LIN {X 0,Y 249.072,Z 125.772,A -85,B 0,C 180,E1 -19026.339,E2 -19026.339} C_VEL
LIN {X 0,Y 249.004,Z 125.778,A -85,B 0,C 180,E1 -19030.813,E2 -19030.813} C_VEL
LIN {X 0,Y 250.137,Z 128.804,A -85,B 0,C 180,E1 -19031.188,E2 -19031.188} C_VEL
LIN {X 0,Y 258.788,Z 144.824,A -85,B 0,C 180,E1 -19033.307,E2 -19033.307} C_VEL
LIN {X 0,Y 270.836,Z 168.303,A -85,B 0,C 180,E1 -19036.063,E2 -19036.063} C_VEL
LIN {X 0,Y 280.754,Z 188.589,A -85,B 0,C 180,E1 -19038.178,E2 -19038.178} C_VEL
LIN {X 0,Y 271.037,Z 309.257,A -85,B 0,C 180,E1 -19042.807,E2 -19042.807} C_VEL
LIN {X 0,Y 269.496,Z 326.293,A -85,B 0,C 180,E1 -19043.763,E2 -19043.763} C_VEL
LIN {X 0,Y 267.518,Z 343.702,A -85,B 0,C 180,E1 -19045.037,E2 -19045.037} C_VEL
LIN {X 0,Y 265.194,Z 361.036,A -85,B 0,C 180,E1 -19046.64,E2 -19046.64} C_VEL
LIN {X 0,Y 262.588,Z 377.74,A -85,B 0,C 180,E1 -19048.54,E2 -19048.54} C_VEL
LIN {X 0,Y 259.925,Z 393.091,A -85,B 0,C 180,E1 -19050.654,E2 -19050.654} C_VEL
LIN {X 0,Y 257.421,Z 407.3,A -85,B 0,C 180,E1 -19053.006,E2 -19053.006} C_VEL
LIN {X 0,Y 254.978,Z 420.401,A -85,B 0,C 180,E1 -19055.578,E2 -19055.578} C_VEL
LIN {X 0,Y 252.965,Z 432.478,A -85,B 0,C 180,E1 -19058.4,E2 -19058.4} C_VEL
LIN {X 0,Y 251.134,Z 442.727,A -85,B 0,C 180,E1 -19061.226,E2 -19061.226} C_VEL
LIN {X 0,Y 249.859,Z 451.559,A -85,B 0,C 180,E1 -19064.083,E2 -19064.083} C_VEL
LIN {X 0,Y 248.75,Z 459.037,A -85,B 0,C 180,E1 -19066.937,E2 -19066.937} C_VEL
LIN {X 0,Y 248.058,Z 466.178,A -85,B 0,C 180,E1 -19070.212,E2 -19070.212} C_VEL
LIN {X 0,Y 247.625,Z 471.999,A -85,B 0,C 180,E1 -19073.481,E2 -19073.481} C_VEL
LIN {X 0,Y 247.502,Z 476.6,A -85,B 0,C 180,E1 -19076.744,E2 -19076.744} C_VEL
LIN {X 0,Y 247.516,Z 480.03,A -85,B 0,C 180,E1 -19080,E2 -19080} C_VEL
LIN {X 0,Y 247.605,Z 480.817,A -85,B 0,C 180,E1 -19080.95,E2 -19080.95} C_VEL
LIN {X 0,Y 247.405,Z 481.54,A -85,B 0,C 180,E1 -19081.844,E2 -19081.844} C_VEL
LIN {X 0,Y 245.705,Z 482.796,A -85,B 0,C 180,E1 -19083.616,E2 -19083.616} C_VEL
LIN {X 0,Y 242.493,Z 484.244,A -85,B 0,C 180,E1 -19086.303,E2 -19086.303} C_VEL
LIN {X 0,Y 241.835,Z 484.743,A -85,B 0,C 180,E1 -19087.697,E2 -19087.697} C_VEL
LIN {X 0,Y 241.906,Z 484.875,A -85,B 0,C 180,E1 -19088.165,E2 -19088.165} C_VEL
LIN {X 0,Y 243.543,Z 485.077,A -85,B 0,C 180,E1 -19091.654,E2 -19091.654} C_VEL
LIN {X 0,Y 245.526,Z 484.42,A -85,B 0,C 180,E1 -19094.929,E2 -19094.929} C_VEL
LIN {X 0,Y 248.17,Z 482.778,A -85,B 0,C 180,E1 -19098.15,E2 -19098.15} C_VEL
LIN {X 0,Y 251.479,Z 480.342,A -85,B 0,C 180,E1 -19101.303,E2 -19101.303} C_VEL
LIN {X 0,Y 256.919,Z 475.829,A -85,B 0,C 180,E1 -19105.19,E2 -19105.19} C_VEL
LIN {X 0,Y 263.085,Z 470.156,A -85,B 0,C 180,E1 -19108.741,E2 -19108.741} C_VEL
LIN {X 0,Y 270.575,Z 462.894,A -85,B 0,C 180,E1 -19112.172,E2 -19112.172} C_VEL
LIN {X 0,Y 279.123,Z 454.142,A -85,B 0,C 180,E1 -19115.388,E2 -19115.388} C_VEL
LIN {X 0,Y 288.335,Z 444.274,A -85,B 0,C 180,E1 -19118.206,E2 -19118.206} C_VEL
LIN {X 0,Y 299.61,Z 431.582,A -85,B 0,C 180,E1 -19121.056,E2 -19121.056} C_VEL
LIN {X 0,Y 308.942,Z 420.434,A -85,B 0,C 180,E1 -19123.036,E2 -19123.036} C_VEL
LIN {X 0,Y 310.463,Z 418.647,A -85,B 0,C 180,E1 -19123.581,E2 -19123.581} C_VEL
LIN {X 0,Y 299.973,Z 432.572,A -85,B 0,C 180,E1 -19125.342,E2 -19125.342} C_VEL
LIN {X 0,Y 289.18,Z 446.505,A -85,B 0,C 180,E1 -19127.59,E2 -19127.59} C_VEL
LIN {X 0,Y 279.364,Z 458.973,A -85,B 0,C 180,E1 -19130.095,E2 -19130.095} C_VEL
LIN {X 0,Y 269.8,Z 471.184,A -85,B 0,C 180,E1 -19133.192,E2 -19133.192} C_VEL
LIN {X 0,Y 261.449,Z 481.983,A -85,B 0,C 180,E1 -19136.623,E2 -19136.623} C_VEL
LIN {X 0,Y 255.897,Z 489.259,A -85,B 0,C 180,E1 -19139.462,E2 -19139.462} C_VEL
LIN {X 0,Y 250.118,Z 497.302,A -85,B 0,C 180,E1 -19143.282,E2 -19143.282} C_VEL
LIN {X 0,Y 245.702,Z 503.944,A -85,B 0,C 180,E1 -19147.284,E2 -19147.284} C_VEL
LIN {X 0,Y 242.612,Z 509.118,A -85,B 0,C 180,E1 -19151.418,E2 -19151.418} C_VEL
LIN {X 0,Y 241.094,Z 512.285,A -85,B 0,C 180,E1 -19154.789,E2 -19154.789} C_VEL
LIN {X 0,Y 240.168,Z 514.482,A -85,B 0,C 180,E1 -19158.179,E2 -19158.179} C_VEL
LIN {X 0,Y 240.048,Z 515.814,A -85,B 0,C 180,E1 -19161.581,E2 -19161.581} C_VEL
LIN {X 0,Y 240.331,Z 516.045,A -85,B 0,C 180,E1 -19164.966,E2 -19164.966} C_VEL
LIN {X 0,Y 240.652,Z 515.281,A -85,B 0,C 180,E1 -19168.325,E2 -19168.325} C_VEL
LIN {X 0,Y 240.951,Z 514.432,A -85,B 0,C 180,E1 -19169.999,E2 -19169.999} C_VEL
LIN {X 0,Y 240.777,Z 511.777,A -85,B 0,C 180,E1 -19173.346,E2 -19173.346} C_VEL
LIN {X 0,Y 240.774,Z 507.887,A -85,B 0,C 180,E1 -19176.704,E2 -19176.704} C_VEL
LIN {X 0,Y 240.633,Z 502.482,A -85,B 0,C 180,E1 -19180.091,E2 -19180.091} C_VEL
LIN {X 0,Y 240.972,Z 495.645,A -85,B 0,C 180,E1 -19183.492,E2 -19183.492} C_VEL
LIN {X 0,Y 241.793,Z 487.201,A -85,B 0,C 180,E1 -19186.896,E2 -19186.896} C_VEL
LIN {X 0,Y 242.929,Z 478.349,A -85,B 0,C 180,E1 -19189.871,E2 -19189.871} C_VEL
LIN {X 0,Y 244.802,Z 466.818,A -85,B 0,C 180,E1 -19193.097,E2 -19193.097} C_VEL
LIN {X 0,Y 247.146,Z 453.598,A -85,B 0,C 180,E1 -19196.152,E2 -19196.152} C_VEL
LIN {X 0,Y 249.783,Z 439.422,A -85,B 0,C 180,E1 -19198.866,E2 -19198.866} C_VEL
LIN {X 0,Y 252.637,Z 424.677,A -85,B 0,C 180,E1 -19201.205,E2 -19201.205} C_VEL
LIN {X 0,Y 255.625,Z 408.15,A -85,B 0,C 180,E1 -19203.357,E2 -19203.357} C_VEL
LIN {X 0,Y 258.348,Z 392.121,A -85,B 0,C 180,E1 -19205.057,E2 -19205.057} C_VEL
LIN {X 0,Y 261.07,Z 374.354,A -85,B 0,C 180,E1 -19206.554,E2 -19206.554} C_VEL
LIN {X 0,Y 263.379,Z 357.048,A -85,B 0,C 180,E1 -19207.677,E2 -19207.677} C_VEL
LIN {X 0,Y 265.064,Z 339.199,A -85,B 0,C 180,E1 -19208.541,E2 -19208.541} C_VEL
LIN {X 0,Y 276.313,Z 206.857,A -85,B 0,C 180,E1 -19213.748,E2 -19213.748} C_VEL
LIN {X 0,Y 275.816,Z 204.209,A -85,B 0,C 180,E1 -19213.93,E2 -19213.93} C_VEL
LIN {X 0,Y 262.961,Z 174.544,A -85,B 0,C 180,E1 -19216.972,E2 -19216.972} C_VEL
LIN {X 0,Y 252.135,Z 150.966,A -85,B 0,C 180,E1 -19219.735,E2 -19219.735} C_VEL
LIN {X 0,Y 245.805,Z 137.764,A -85,B 0,C 180,E1 -19221.482,E2 -19221.482} C_VEL
LIN {X 0,Y 242.032,Z 126.649,A -85,B 0,C 180,E1 -19224.497,E2 -19224.497} C_VEL
LIN {X 0,Y 241.972,Z 126.656,A -85,B 0,C 180,E1 -19228.48,E2 -19228.48} C_VEL
LIN {X 0,Y 242.003,Z 126.657,A -85,B 0,C 180,E1 -19232.312,E2 -19232.312} C_VEL
LIN {X 0,Y 242.053,Z 126.649,A -85,B 0,C 180,E1 -19236.016,E2 -19236.016} C_VEL
LIN {X 0,Y 242.033,Z 126.649,A -85,B 0,C 180,E1 -19239.608,E2 -19239.608} C_VEL
LIN {X 0,Y 242.159,Z 126.63,A -85,B 0,C 180,E1 -19243.278,E2 -19243.278} C_VEL
LIN {X 0,Y 242.183,Z 126.624,A -85,B 0,C 180,E1 -19248.28,E2 -19248.28} C_VEL
LIN {X 0,Y 242.431,Z 126.602,A -85,B 0,C 180,E1 -19251.666,E2 -19251.666} C_VEL
LIN {X 0,Y 242.257,Z 126.611,A -85,B 0,C 180,E1 -19255.007,E2 -19255.007} C_VEL
LIN {X 0,Y 242.633,Z 126.573,A -85,B 0,C 180,E1 -19258.34,E2 -19258.34} C_VEL
LIN {X 0,Y 242.633,Z 126.573,A -85,B 0,C 180,E1 -19261.66,E2 -19261.66} C_VEL
LIN {X 0,Y 242.426,Z 126.595,A -85,B 0,C 180,E1 -19266.735,E2 -19266.735} C_VEL
LIN {X 0,Y 242.342,Z 126.608,A -85,B 0,C 180,E1 -19270.021,E2 -19270.021} C_VEL
LIN {X 0,Y 242.163,Z 126.634,A -85,B 0,C 180,E1 -19275.141,E2 -19275.141} C_VEL
LIN {X 0,Y 242.069,Z 126.64,A -85,B 0,C 180,E1 -19278.625,E2 -19278.625} C_VEL
LIN {X 0,Y 242.009,Z 126.649,A -85,B 0,C 180,E1 -19282.18,E2 -19282.18} C_VEL
LIN {X 0,Y 242.063,Z 126.643,A -85,B 0,C 180,E1 -19285.839,E2 -19285.839} C_VEL
LIN {X 0,Y 242.026,Z 126.646,A -85,B 0,C 180,E1 -19289.581,E2 -19289.581} C_VEL
LIN {X 0,Y 241.977,Z 126.655,A -85,B 0,C 180,E1 -19293.493,E2 -19293.493} C_VEL
LIN {X 0,Y 241.985,Z 126.649,A -85,B 0,C 180,E1 -19297.583,E2 -19297.583} C_VEL
LIN {X 0,Y 241.936,Z 126.659,A -85,B 0,C 180,E1 -19301.923,E2 -19301.923} C_VEL
LIN {X 0,Y 241.942,Z 126.654,A -85,B 0,C 180,E1 -19306.569,E2 -19306.569} C_VEL
LIN {X 0,Y 241.986,Z 126.653,A -85,B 0,C 180,E1 -19310.288,E2 -19310.288} C_VEL
LIN {X 0,Y 242.035,Z 126.643,A -85,B 0,C 180,E1 -19314.499,E2 -19314.499} C_VEL
LIN {X 0,Y 241.974,Z 126.657,A -85,B 0,C 180,E1 -19318.481,E2 -19318.481} C_VEL
LIN {X 0,Y 242.005,Z 126.647,A -85,B 0,C 180,E1 -19322.314,E2 -19322.314} C_VEL
LIN {X 0,Y 242.059,Z 126.645,A -85,B 0,C 180,E1 -19326.017,E2 -19326.017} C_VEL
LIN {X 0,Y 242.06,Z 126.64,A -85,B 0,C 180,E1 -19329.611,E2 -19329.611} C_VEL
LIN {X 0,Y 242.163,Z 126.63,A -85,B 0,C 180,E1 -19333.279,E2 -19333.279} C_VEL
LIN {X 0,Y 242.187,Z 126.632,A -85,B 0,C 180,E1 -19338.281,E2 -19338.281} C_VEL
LIN {X 0,Y 242.436,Z 126.594,A -85,B 0,C 180,E1 -19341.667,E2 -19341.667} C_VEL
LIN {X 0,Y 242.261,Z 126.618,A -85,B 0,C 180,E1 -19345.008,E2 -19345.008} C_VEL
LIN {X 0,Y 242.637,Z 126.574,A -85,B 0,C 180,E1 -19348.341,E2 -19348.341} C_VEL
LIN {X 0,Y 242.637,Z 126.571,A -85,B 0,C 180,E1 -19351.661,E2 -19351.661} C_VEL
LIN {X 0,Y 242.436,Z 126.598,A -85,B 0,C 180,E1 -19356.66,E2 -19356.66} C_VEL
LIN {X 0,Y 242.348,Z 126.607,A -85,B 0,C 180,E1 -19360.021,E2 -19360.021} C_VEL
LIN {X 0,Y 242.169,Z 126.633,A -85,B 0,C 180,E1 -19365.142,E2 -19365.142} C_VEL
LIN {X 0,Y 242.076,Z 126.638,A -85,B 0,C 180,E1 -19368.625,E2 -19368.625} C_VEL
LIN {X 0,Y 242.017,Z 126.647,A -85,B 0,C 180,E1 -19372.181,E2 -19372.181} C_VEL
LIN {X 0,Y 242.069,Z 126.645,A -85,B 0,C 180,E1 -19375.839,E2 -19375.839} C_VEL
LIN {X 0,Y 242.032,Z 126.653,A -85,B 0,C 180,E1 -19379.581,E2 -19379.581} C_VEL
LIN {X 0,Y 241.994,Z 126.656,A -85,B 0,C 180,E1 -19383.492,E2 -19383.492} C_VEL
LIN {X 0,Y 242.006,Z 126.65,A -85,B 0,C 180,E1 -19387.58,E2 -19387.58} C_VEL
LIN {X 0,Y 241.947,Z 126.657,A -85,B 0,C 180,E1 -19389.791,E2 -19389.791} C_VEL
LIN {X 0,Y 242.99,Z 129.564,A -85,B 0,C 180,E1 -19390.134,E2 -19390.134} C_VEL
LIN {X 0,Y 244.338,Z 131.856,A -85,B 0,C 180,E1 -19390.479,E2 -19390.479} C_VEL
LIN {X 0,Y 254.963,Z 151.723,A -85,B 0,C 180,E1 -19393.154,E2 -19393.154} C_VEL
LIN {X 0,Y 267.479,Z 176.469,A -85,B 0,C 180,E1 -19396.064,E2 -19396.064} C_VEL
LIN {X 0,Y 274.342,Z 190.869,A -85,B 0,C 180,E1 -19397.576,E2 -19397.576} C_VEL
LIN {X 0,Y 264.433,Z 309.481,A -85,B 0,C 180,E1 -19402.257,E2 -19402.257} C_VEL
LIN {X 0,Y 262.786,Z 327.136,A -85,B 0,C 180,E1 -19403.28,E2 -19403.28} C_VEL
LIN {X 0,Y 260.733,Z 344.437,A -85,B 0,C 180,E1 -19404.583,E2 -19404.583} C_VEL
LIN {X 0,Y 258.512,Z 360.775,A -85,B 0,C 180,E1 -19406.129,E2 -19406.129} C_VEL
LIN {X 0,Y 255.822,Z 377.614,A -85,B 0,C 180,E1 -19408.073,E2 -19408.073} C_VEL
LIN {X 0,Y 253.1,Z 393.039,A -85,B 0,C 180,E1 -19410.241,E2 -19410.241} C_VEL
LIN {X 0,Y 250.503,Z 407.312,A -85,B 0,C 180,E1 -19412.651,E2 -19412.651} C_VEL
LIN {X 0,Y 247.9,Z 421.11,A -85,B 0,C 180,E1 -19415.426,E2 -19415.426} C_VEL
LIN {X 0,Y 245.912,Z 432.635,A -85,B 0,C 180,E1 -19418.19,E2 -19418.19} C_VEL
LIN {X 0,Y 244.055,Z 442.978,A -85,B 0,C 180,E1 -19421.097,E2 -19421.097} C_VEL
LIN {X 0,Y 242.733,Z 451.861,A -85,B 0,C 180,E1 -19424.034,E2 -19424.034} C_VEL
LIN {X 0,Y 241.529,Z 460.386,A -85,B 0,C 180,E1 -19427.394,E2 -19427.394} C_VEL
LIN {X 0,Y 240.858,Z 467.389,A -85,B 0,C 180,E1 -19430.765,E2 -19430.765} C_VEL
LIN {X 0,Y 240.452,Z 473.046,A -85,B 0,C 180,E1 -19434.11,E2 -19434.11} C_VEL
LIN {X 0,Y 240.426,Z 476.555,A -85,B 0,C 180,E1 -19436.648,E2 -19436.648} C_VEL
LIN {X 0,Y 240.425,Z 480.217,A -85,B 0,C 180,E1 -19440,E2 -19440} C_VEL
LIN {X 0,Y 240.885,Z 482.815,A -85,B 0,C 180,E1 -19443.345,E2 -19443.345} C_VEL
LIN {X 0,Y 241.482,Z 484.438,A -85,B 0,C 180,E1 -19446.685,E2 -19446.685} C_VEL
LIN {X 0,Y 241.906,Z 484.875,A -85,B 0,C 180,E1 -19448.165,E2 -19448.165} C_VEL
LIN {X 0,Y 241.779,Z 485.264,A -85,B 0,C 180,E1 -19449.562,E2 -19449.562} C_VEL
LIN {X 0,Y 240.042,Z 485.702,A -85,B 0,C 180,E1 -19451.882,E2 -19451.882} C_VEL
LIN {X 0,Y 238.742,Z 485.726,A -85,B 0,C 180,E1 -19453.762,E2 -19453.762} C_VEL
LIN {X 0,Y 238.672,Z 485.475,A -85,B 0,C 180,E1 -19455.183,E2 -19455.183} C_VEL
LIN {X 0,Y 238.933,Z 485.329,A -85,B 0,C 180,E1 -19455.652,E2 -19455.652} C_VEL
LIN {X 0,Y 243.189,Z 483.096,A -85,B 0,C 180,E1 -19460.291,E2 -19460.291} C_VEL
LIN {X 0,Y 247.128,Z 480.38,A -85,B 0,C 180,E1 -19463.462,E2 -19463.462} C_VEL
LIN {X 0,Y 253.4,Z 475.577,A -85,B 0,C 180,E1 -19467.435,E2 -19467.435} C_VEL
LIN {X 0,Y 260.197,Z 469.904,A -85,B 0,C 180,E1 -19470.877,E2 -19470.877} C_VEL
LIN {X 0,Y 268.479,Z 462.552,A -85,B 0,C 180,E1 -19474.25,E2 -19474.25} C_VEL
LIN {X 0,Y 277.871,Z 453.719,A -85,B 0,C 180,E1 -19477.374,E2 -19477.374} C_VEL
LIN {X 0,Y 287.282,Z 444.421,A -85,B 0,C 180,E1 -19479.954,E2 -19479.954} C_VEL
LIN {X 0,Y 298.648,Z 432.545,A -85,B 0,C 180,E1 -19482.576,E2 -19482.576} C_VEL
LIN {X 0,Y 301.527,Z 429.387,A -85,B 0,C 180,E1 -19483.167,E2 -19483.167} C_VEL
LIN {X 0,Y 300.71,Z 430.48,A -85,B 0,C 180,E1 -19483.571,E2 -19483.571} C_VEL
LIN {X 0,Y 289.203,Z 444.239,A -85,B 0,C 180,E1 -19485.679,E2 -19485.679} C_VEL
LIN {X 0,Y 278.639,Z 456.594,A -85,B 0,C 180,E1 -19488.055,E2 -19488.055} C_VEL
LIN {X 0,Y 269.174,Z 467.539,A -85,B 0,C 180,E1 -19490.715,E2 -19490.715} C_VEL
LIN {X 0,Y 259.872,Z 478.33,A -85,B 0,C 180,E1 -19493.969,E2 -19493.969} C_VEL
LIN {X 0,Y 252.646,Z 486.874,A -85,B 0,C 180,E1 -19497.149,E2 -19497.149} C_VEL
LIN {X 0,Y 246.081,Z 495.016,A -85,B 0,C 180,E1 -19500.953,E2 -19500.953} C_VEL
LIN {X 0,Y 241.207,Z 501.217,A -85,B 0,C 180,E1 -19504.587,E2 -19504.587} C_VEL
LIN {X 0,Y 236.913,Z 507.236,A -85,B 0,C 180,E1 -19509.145,E2 -19509.145} C_VEL
LIN {X 0,Y 234.429,Z 511.459,A -85,B 0,C 180,E1 -19513.603,E2 -19513.603} C_VEL
LIN {X 0,Y 233.137,Z 514.042,A -85,B 0,C 180,E1 -19517.817,E2 -19517.817} C_VEL
LIN {X 0,Y 232.96,Z 515.129,A -85,B 0,C 180,E1 -19521.323,E2 -19521.323} C_VEL
LIN {X 0,Y 233.27,Z 515.257,A -85,B 0,C 180,E1 -19524.813,E2 -19524.813} C_VEL
LIN {X 0,Y 233.636,Z 514.3,A -85,B 0,C 180,E1 -19528.275,E2 -19528.275} C_VEL
LIN {X 0,Y 233.913,Z 513.44,A -85,B 0,C 180,E1 -19529.999,E2 -19529.999} C_VEL
LIN {X 0,Y 233.753,Z 510.574,A -85,B 0,C 180,E1 -19533.446,E2 -19533.446} C_VEL
LIN {X 0,Y 233.747,Z 506.487,A -85,B 0,C 180,E1 -19536.906,E2 -19536.906} C_VEL
LIN {X 0,Y 233.617,Z 500.93,A -85,B 0,C 180,E1 -19540.398,E2 -19540.398} C_VEL
LIN {X 0,Y 234.009,Z 493.845,A -85,B 0,C 180,E1 -19543.901,E2 -19543.901} C_VEL
LIN {X 0,Y 234.905,Z 485.132,A -85,B 0,C 180,E1 -19547.407,E2 -19547.407} C_VEL
LIN {X 0,Y 236.107,Z 475.965,A -85,B 0,C 180,E1 -19550.471,E2 -19550.471} C_VEL
LIN {X 0,Y 237.947,Z 465.069,A -85,B 0,C 180,E1 -19553.536,E2 -19553.536} C_VEL
LIN {X 0,Y 240.244,Z 452.502,A -85,B 0,C 180,E1 -19556.493,E2 -19556.493} C_VEL
LIN {X 0,Y 242.677,Z 439.747,A -85,B 0,C 180,E1 -19559.017,E2 -19559.017} C_VEL
LIN {X 0,Y 245.628,Z 424.816,A -85,B 0,C 180,E1 -19561.477,E2 -19561.477} C_VEL
LIN {X 0,Y 248.653,Z 408.492,A -85,B 0,C 180,E1 -19563.688,E2 -19563.688} C_VEL
LIN {X 0,Y 251.446,Z 392.494,A -85,B 0,C 180,E1 -19565.447,E2 -19565.447} C_VEL
LIN {X 0,Y 254.246,Z 374.872,A -85,B 0,C 180,E1 -19566.992,E2 -19566.992} C_VEL
LIN {X 0,Y 256.732,Z 356.781,A -85,B 0,C 180,E1 -19568.205,E2 -19568.205} C_VEL
LIN {X 0,Y 258.446,Z 339.216,A -85,B 0,C 180,E1 -19569.089,E2 -19569.089} C_VEL
LIN {X 0,Y 270.009,Z 207.635,A -85,B 0,C 180,E1 -19574.425,E2 -19574.425} C_VEL
LIN {X 0,Y 257.52,Z 178.451,A -85,B 0,C 180,E1 -19577.486,E2 -19577.486} C_VEL
LIN {X 0,Y 245.86,Z 153.121,A -85,B 0,C 180,E1 -19580.544,E2 -19580.544} C_VEL
LIN {X 0,Y 238.279,Z 137.255,A -85,B 0,C 180,E1 -19582.705,E2 -19582.705} C_VEL
LIN {X 0,Y 234.94,Z 127.532,A -85,B 0,C 180,E1 -19585.417,E2 -19585.417} C_VEL
LIN {X 0,Y 234.928,Z 127.535,A -85,B 0,C 180,E1 -19589.432,E2 -19589.432} C_VEL
LIN {X 0,Y 234.99,Z 127.528,A -85,B 0,C 180,E1 -19593.793,E2 -19593.793} C_VEL
LIN {X 0,Y 235.007,Z 127.524,A -85,B 0,C 180,E1 -19598.97,E2 -19598.97} C_VEL
LIN {X 0,Y 235.092,Z 127.51,A -85,B 0,C 180,E1 -19603.059,E2 -19603.059} C_VEL
LIN {X 0,Y 235.143,Z 127.5,A -85,B 0,C 180,E1 -19607.924,E2 -19607.924} C_VEL
LIN {X 0,Y 235.386,Z 127.478,A -85,B 0,C 180,E1 -19611.415,E2 -19611.415} C_VEL
LIN {X 0,Y 235.402,Z 127.473,A -85,B 0,C 180,E1 -19613.141,E2 -19613.141} C_VEL
LIN {X 0,Y 235.592,Z 127.451,A -85,B 0,C 180,E1 -19618.291,E2 -19618.291} C_VEL
LIN {X 0,Y 235.592,Z 127.45,A -85,B 0,C 180,E1 -19621.71,E2 -19621.71} C_VEL
LIN {X 0,Y 235.402,Z 127.471,A -85,B 0,C 180,E1 -19626.859,E2 -19626.859} C_VEL
LIN {X 0,Y 235.249,Z 127.491,A -85,B 0,C 180,E1 -19630.326,E2 -19630.326} C_VEL
LIN {X 0,Y 235.11,Z 127.51,A -85,B 0,C 180,E1 -19635.607,E2 -19635.607} C_VEL
LIN {X 0,Y 235.005,Z 127.523,A -85,B 0,C 180,E1 -19639.206,E2 -19639.206} C_VEL
LIN {X 0,Y 234.957,Z 127.529,A -85,B 0,C 180,E1 -19642.883,E2 -19642.883} C_VEL
LIN {X 0,Y 234.966,Z 127.527,A -85,B 0,C 180,E1 -19646.658,E2 -19646.658} C_VEL
LIN {X 0,Y 234.928,Z 127.53,A -85,B 0,C 180,E1 -19650.568,E2 -19650.568} C_VEL
LIN {X 0,Y 234.926,Z 127.534,A -85,B 0,C 180,E1 -19654.639,E2 -19654.639} C_VEL
LIN {X 0,Y 234.938,Z 127.527,A -85,B 0,C 180,E1 -19658.945,E2 -19658.945} C_VEL
LIN {X 0,Y 234.888,Z 127.537,A -85,B 0,C 180,E1 -19663.486,E2 -19663.486} C_VEL
LIN {X 0,Y 234.92,Z 127.529,A -85,B 0,C 180,E1 -19666.523,E2 -19666.523} C_VEL
LIN {X 0,Y 234.952,Z 127.529,A -85,B 0,C 180,E1 -19671.087,E2 -19671.087} C_VEL
LIN {X 0,Y 234.959,Z 127.526,A -85,B 0,C 180,E1 -19675.368,E2 -19675.368} C_VEL
LIN {X 0,Y 234.967,Z 127.527,A -85,B 0,C 180,E1 -19680.159,E2 -19680.159} C_VEL
LIN {X 0,Y 234.993,Z 127.523,A -85,B 0,C 180,E1 -19683.795,E2 -19683.795} C_VEL
LIN {X 0,Y 235.027,Z 127.517,A -85,B 0,C 180,E1 -19688.973,E2 -19688.973} C_VEL
LIN {X 0,Y 235.096,Z 127.511,A -85,B 0,C 180,E1 -19693.06,E2 -19693.06} C_VEL
LIN {X 0,Y 235.119,Z 127.51,A -85,B 0,C 180,E1 -19697.923,E2 -19697.923} C_VEL
LIN {X 0,Y 235.391,Z 127.47,A -85,B 0,C 180,E1 -19701.416,E2 -19701.416} C_VEL
LIN {X 0,Y 235.406,Z 127.472,A -85,B 0,C 180,E1 -19703.143,E2 -19703.143} C_VEL
LIN {X 0,Y 235.597,Z 127.452,A -85,B 0,C 180,E1 -19708.292,E2 -19708.292} C_VEL
LIN {X 0,Y 235.597,Z 127.447,A -85,B 0,C 180,E1 -19711.711,E2 -19711.711} C_VEL
LIN {X 0,Y 235.407,Z 127.473,A -85,B 0,C 180,E1 -19716.86,E2 -19716.86} C_VEL
LIN {X 0,Y 235.255,Z 127.488,A -85,B 0,C 180,E1 -19720.327,E2 -19720.327} C_VEL
LIN {X 0,Y 235.116,Z 127.514,A -85,B 0,C 180,E1 -19725.607,E2 -19725.607} C_VEL
LIN {X 0,Y 235.012,Z 127.518,A -85,B 0,C 180,E1 -19729.206,E2 -19729.206} C_VEL
LIN {X 0,Y 234.965,Z 127.524,A -85,B 0,C 180,E1 -19732.884,E2 -19732.884} C_VEL
LIN {X 0,Y 234.972,Z 127.527,A -85,B 0,C 180,E1 -19736.658,E2 -19736.658} C_VEL
LIN {X 0,Y 234.935,Z 127.533,A -85,B 0,C 180,E1 -19740.569,E2 -19740.569} C_VEL
LIN {X 0,Y 234.964,Z 127.527,A -85,B 0,C 180,E1 -19744.634,E2 -19744.634} C_VEL
LIN {X 0,Y 234.947,Z 127.559,A -85,B 0,C 180,E1 -19748.72,E2 -19748.72} C_VEL
LIN {X 0,Y 235.955,Z 130.389,A -85,B 0,C 180,E1 -19749.062,E2 -19749.062} C_VEL
LIN {X 0,Y 244.618,Z 146.212,A -85,B 0,C 180,E1 -19751.362,E2 -19751.362} C_VEL
LIN {X 0,Y 257.248,Z 170.753,A -85,B 0,C 180,E1 -19754.486,E2 -19754.486} C_VEL
LIN {X 0,Y 267.827,Z 192.409,A -85,B 0,C 180,E1 -19756.899,E2 -19756.899} C_VEL
LIN {X 0,Y 265.441,Z 220.63,A -85,B 0,C 180,E1 -19758.024,E2 -19758.024} C_VEL
LIN {X 0,Y 257.797,Z 310.244,A -85,B 0,C 180,E1 -19761.719,E2 -19761.719} C_VEL
LIN {X 0,Y 256.17,Z 326.998,A -85,B 0,C 180,E1 -19762.715,E2 -19762.715} C_VEL
LIN {X 0,Y 253.984,Z 345.031,A -85,B 0,C 180,E1 -19764.106,E2 -19764.106} C_VEL
LIN {X 0,Y 251.537,Z 362.229,A -85,B 0,C 180,E1 -19765.785,E2 -19765.785} C_VEL
LIN {X 0,Y 248.775,Z 379.205,A -85,B 0,C 180,E1 -19767.829,E2 -19767.829} C_VEL
LIN {X 0,Y 246.01,Z 394.186,A -85,B 0,C 180,E1 -19770.004,E2 -19770.004} C_VEL
LIN {X 0,Y 243.379,Z 408.38,A -85,B 0,C 180,E1 -19772.482,E2 -19772.482} C_VEL
LIN {X 0,Y 240.929,Z 421.124,A -85,B 0,C 180,E1 -19775.126,E2 -19775.126} C_VEL
LIN {X 0,Y 238.886,Z 432.733,A -85,B 0,C 180,E1 -19777.969,E2 -19777.969} C_VEL
LIN {X 0,Y 236.837,Z 444.198,A -85,B 0,C 180,E1 -19781.294,E2 -19781.294} C_VEL
LIN {X 0,Y 235.411,Z 453.238,A -85,B 0,C 180,E1 -19784.414,E2 -19784.414} C_VEL
LIN {X 0,Y 234.316,Z 461.645,A -85,B 0,C 180,E1 -19787.88,E2 -19787.88} C_VEL
LIN {X 0,Y 233.717,Z 468.561,A -85,B 0,C 180,E1 -19791.352,E2 -19791.352} C_VEL
LIN {X 0,Y 233.342,Z 474.121,A -85,B 0,C 180,E1 -19794.816,E2 -19794.816} C_VEL
LIN {X 0,Y 233.288,Z 478.56,A -85,B 0,C 180,E1 -19798.273,E2 -19798.273} C_VEL
LIN {X 0,Y 233.53,Z 481.851,A -85,B 0,C 180,E1 -19801.724,E2 -19801.724} C_VEL
LIN {X 0,Y 234.096,Z 484.152,A -85,B 0,C 180,E1 -19805.167,E2 -19805.167} C_VEL
LIN {X 0,Y 234.967,Z 485.508,A -85,B 0,C 180,E1 -19808.601,E2 -19808.601} C_VEL
LIN {X 0,Y 236.623,Z 485.909,A -85,B 0,C 180,E1 -19812,E2 -19812} C_VEL
LIN {X 0,Y 238.933,Z 485.329,A -85,B 0,C 180,E1 -19815.652,E2 -19815.652} C_VEL
LIN {X 0,Y 239.382,Z 484.966,A -85,B 0,C 180,E1 -19817.061,E2 -19817.061} C_VEL
LIN {X 0,Y 238.676,Z 484.454,A -85,B 0,C 180,E1 -19819.432,E2 -19819.432} C_VEL
LIN {X 0,Y 238.397,Z 483.717,A -85,B 0,C 180,E1 -19821.803,E2 -19821.803} C_VEL
LIN {X 0,Y 239.491,Z 482.826,A -85,B 0,C 180,E1 -19823.176,E2 -19823.176} C_VEL
LIN {X 0,Y 245.746,Z 478.777,A -85,B 0,C 180,E1 -19827.231,E2 -19827.231} C_VEL
LIN {X 0,Y 252.964,Z 473.532,A -85,B 0,C 180,E1 -19830.929,E2 -19830.929} C_VEL
LIN {X 0,Y 261.329,Z 466.956,A -85,B 0,C 180,E1 -19834.385,E2 -19834.385} C_VEL
LIN {X 0,Y 270.832,Z 458.986,A -85,B 0,C 180,E1 -19837.576,E2 -19837.576} C_VEL
LIN {X 0,Y 281.474,Z 449.55,A -85,B 0,C 180,E1 -19840.48,E2 -19840.48} C_VEL
LIN {X 0,Y 292.923,Z 438.77,A -85,B 0,C 180,E1 -19843.052,E2 -19843.052} C_VEL
LIN {X 0,Y 292.366,Z 439.463,A -85,B 0,C 180,E1 -19843.341,E2 -19843.341} C_VEL
LIN {X 0,Y 280.864,Z 451.884,A -85,B 0,C 180,E1 -19845.521,E2 -19845.521} C_VEL
LIN {X 0,Y 269.258,Z 464.188,A -85,B 0,C 180,E1 -19848.272,E2 -19848.272} C_VEL
LIN {X 0,Y 259.008,Z 475.066,A -85,B 0,C 180,E1 -19851.384,E2 -19851.384} C_VEL
LIN {X 0,Y 248.336,Z 486.343,A -85,B 0,C 180,E1 -19855.527,E2 -19855.527} C_VEL
LIN {X 0,Y 241.186,Z 494.322,A -85,B 0,C 180,E1 -19859.339,E2 -19859.339} C_VEL
LIN {X 0,Y 235.307,Z 500.964,A -85,B 0,C 180,E1 -19863.383,E2 -19863.383} C_VEL
LIN {X 0,Y 231.691,Z 505.408,A -85,B 0,C 180,E1 -19866.774,E2 -19866.774} C_VEL
LIN {X 0,Y 228.004,Z 510.443,A -85,B 0,C 180,E1 -19872.046,E2 -19872.046} C_VEL
LIN {X 0,Y 226.565,Z 512.697,A -85,B 0,C 180,E1 -19875.63,E2 -19875.63} C_VEL
LIN {X 0,Y 225.901,Z 514.124,A -85,B 0,C 180,E1 -19879.241,E2 -19879.241} C_VEL
LIN {X 0,Y 226.151,Z 514.504,A -85,B 0,C 180,E1 -19883.959,E2 -19883.959} C_VEL
LIN {X 0,Y 226.419,Z 514,A -85,B 0,C 180,E1 -19886.44,E2 -19886.44} C_VEL
LIN {X 0,Y 226.892,Z 512.325,A -85,B 0,C 180,E1 -19889.999,E2 -19889.999} C_VEL
LIN {X 0,Y 226.81,Z 511.019,A -85,B 0,C 180,E1 -19891.774,E2 -19891.774} C_VEL
LIN {X 0,Y 226.725,Z 507.356,A -85,B 0,C 180,E1 -19895.335,E2 -19895.335} C_VEL
LIN {X 0,Y 226.643,Z 503.871,A -85,B 0,C 180,E1 -19897.93,E2 -19897.93} C_VEL
LIN {X 0,Y 226.651,Z 497.553,A -85,B 0,C 180,E1 -19901.627,E2 -19901.627} C_VEL
LIN {X 0,Y 227.248,Z 489.864,A -85,B 0,C 180,E1 -19905.24,E2 -19905.24} C_VEL
LIN {X 0,Y 228.354,Z 480.411,A -85,B 0,C 180,E1 -19908.853,E2 -19908.853} C_VEL
LIN {X 0,Y 229.838,Z 470.538,A -85,B 0,C 180,E1 -19911.997,E2 -19911.997} C_VEL
LIN {X 0,Y 231.899,Z 458.922,A -85,B 0,C 180,E1 -19915.104,E2 -19915.104} C_VEL
LIN {X 0,Y 234.58,Z 445.191,A -85,B 0,C 180,E1 -19918.154,E2 -19918.154} C_VEL
LIN {X 0,Y 237.238,Z 431.741,A -85,B 0,C 180,E1 -19920.65,E2 -19920.65} C_VEL
LIN {X 0,Y 240.258,Z 416.361,A -85,B 0,C 180,E1 -19923.011,E2 -19923.011} C_VEL
LIN {X 0,Y 243.294,Z 400.229,A -85,B 0,C 180,E1 -19925.037,E2 -19925.037} C_VEL
LIN {X 0,Y 246.255,Z 382.596,A -85,B 0,C 180,E1 -19926.82,E2 -19926.82} C_VEL
LIN {X 0,Y 248.768,Z 365.826,A -85,B 0,C 180,E1 -19928.153,E2 -19928.153} C_VEL
LIN {X 0,Y 251.033,Z 347.901,A -85,B 0,C 180,E1 -19929.236,E2 -19929.236} C_VEL
LIN {X 0,Y 262.28,Z 223.969,A -85,B 0,C 180,E1 -19934.496,E2 -19934.496} C_VEL
LIN {X 0,Y 263.554,Z 209.377,A -85,B 0,C 180,E1 -19935.096,E2 -19935.096} C_VEL
LIN {X 0,Y 251.763,Z 181.744,A -85,B 0,C 180,E1 -19938.069,E2 -19938.069} C_VEL
LIN {X 0,Y 240.894,Z 157.856,A -85,B 0,C 180,E1 -19941.018,E2 -19941.018} C_VEL
LIN {X 0,Y 230.756,Z 136.797,A -85,B 0,C 180,E1 -19943.972,E2 -19943.972} C_VEL
LIN {X 0,Y 227.911,Z 128.407,A -85,B 0,C 180,E1 -19946.435,E2 -19946.435} C_VEL
LIN {X 0,Y 227.914,Z 128.409,A -85,B 0,C 180,E1 -19950.437,E2 -19950.437} C_VEL
LIN {X 0,Y 227.924,Z 128.412,A -85,B 0,C 180,E1 -19954.426,E2 -19954.426} C_VEL
LIN {X 0,Y 227.958,Z 128.405,A -85,B 0,C 180,E1 -19958.287,E2 -19958.287} C_VEL
LIN {X 0,Y 228.031,Z 128.389,A -85,B 0,C 180,E1 -19962.825,E2 -19962.825} C_VEL
LIN {X 0,Y 228.09,Z 128.378,A -85,B 0,C 180,E1 -19967.544,E2 -19967.544} C_VEL
LIN {X 0,Y 228.321,Z 128.357,A -85,B 0,C 180,E1 -19971.147,E2 -19971.147} C_VEL
LIN {X 0,Y 228.354,Z 128.351,A -85,B 0,C 180,E1 -19972.929,E2 -19972.929} C_VEL
LIN {X 0,Y 228.551,Z 128.328,A -85,B 0,C 180,E1 -19978.238,E2 -19978.238} C_VEL
LIN {X 0,Y 228.551,Z 128.327,A -85,B 0,C 180,E1 -19981.762,E2 -19981.762} C_VEL
LIN {X 0,Y 228.355,Z 128.349,A -85,B 0,C 180,E1 -19987.072,E2 -19987.072} C_VEL
LIN {X 0,Y 228.168,Z 128.373,A -85,B 0,C 180,E1 -19990.65,E2 -19990.65} C_VEL
LIN {X 0,Y 228.054,Z 128.387,A -85,B 0,C 180,E1 -19996.103,E2 -19996.103} C_VEL
LIN {X 0,Y 227.939,Z 128.404,A -85,B 0,C 180,E1 -19999.826,E2 -19999.826} C_VEL
LIN {X 0,Y 227.91,Z 128.401,A -85,B 0,C 180,E1 -20003.633,E2 -20003.633} C_VEL
LIN {X 0,Y 227.882,Z 128.411,A -85,B 0,C 180,E1 -20007.556,E2 -20007.556} C_VEL
LIN {X 0,Y 227.867,Z 128.408,A -85,B 0,C 180,E1 -20011.623,E2 -20011.623} C_VEL
LIN {X 0,Y 227.877,Z 128.41,A -85,B 0,C 180,E1 -20015.873,E2 -20015.873} C_VEL
LIN {X 0,Y 227.823,Z 128.414,A -85,B 0,C 180,E1 -20020.377,E2 -20020.377} C_VEL
LIN {X 0,Y 227.835,Z 128.411,A -85,B 0,C 180,E1 -20025.192,E2 -20025.192} C_VEL
LIN {X 0,Y 227.872,Z 128.411,A -85,B 0,C 180,E1 -20029.635,E2 -20029.635} C_VEL
LIN {X 0,Y 227.899,Z 128.402,A -85,B 0,C 180,E1 -20034.133,E2 -20034.133} C_VEL
LIN {X 0,Y 227.871,Z 128.413,A -85,B 0,C 180,E1 -20038.379,E2 -20038.379} C_VEL
LIN {X 0,Y 227.884,Z 128.406,A -85,B 0,C 180,E1 -20042.446,E2 -20042.446} C_VEL
LIN {X 0,Y 227.924,Z 128.407,A -85,B 0,C 180,E1 -20046.37,E2 -20046.37} C_VEL
LIN {X 0,Y 227.954,Z 128.399,A -85,B 0,C 180,E1 -20050.177,E2 -20050.177} C_VEL
LIN {X 0,Y 228.058,Z 128.389,A -85,B 0,C 180,E1 -20053.899,E2 -20053.899} C_VEL
LIN {X 0,Y 228.076,Z 128.386,A -85,B 0,C 180,E1 -20057.545,E2 -20057.545} C_VEL
LIN {X 0,Y 228.326,Z 128.35,A -85,B 0,C 180,E1 -20061.148,E2 -20061.148} C_VEL
LIN {X 0,Y 228.359,Z 128.35,A -85,B 0,C 180,E1 -20062.93,E2 -20062.93} C_VEL
LIN {X 0,Y 228.555,Z 128.328,A -85,B 0,C 180,E1 -20068.239,E2 -20068.239} C_VEL
LIN {X 0,Y 228.555,Z 128.323,A -85,B 0,C 180,E1 -20071.763,E2 -20071.763} C_VEL
LIN {X 0,Y 228.36,Z 128.352,A -85,B 0,C 180,E1 -20077.072,E2 -20077.072} C_VEL
LIN {X 0,Y 228.174,Z 128.369,A -85,B 0,C 180,E1 -20080.651,E2 -20080.651} C_VEL
LIN {X 0,Y 228.06,Z 128.389,A -85,B 0,C 180,E1 -20086.103,E2 -20086.103} C_VEL
LIN {X 0,Y 227.946,Z 128.403,A -85,B 0,C 180,E1 -20089.826,E2 -20089.826} C_VEL
LIN {X 0,Y 227.917,Z 128.402,A -85,B 0,C 180,E1 -20093.633,E2 -20093.633} C_VEL
LIN {X 0,Y 227.888,Z 128.408,A -85,B 0,C 180,E1 -20097.556,E2 -20097.556} C_VEL
LIN {X 0,Y 227.876,Z 128.41,A -85,B 0,C 180,E1 -20101.623,E2 -20101.623} C_VEL
LIN {X 0,Y 227.903,Z 128.41,A -85,B 0,C 180,E1 -20105.869,E2 -20105.869} C_VEL
LIN {X 0,Y 227.942,Z 128.468,A -85,B 0,C 180,E1 -20107.591,E2 -20107.591} C_VEL
LIN {X 0,Y 228.933,Z 131.264,A -85,B 0,C 180,E1 -20107.945,E2 -20107.945} C_VEL
LIN {X 0,Y 238.918,Z 149.481,A -85,B 0,C 180,E1 -20110.697,E2 -20110.697} C_VEL
LIN {X 0,Y 252.24,Z 175.591,A -85,B 0,C 180,E1 -20114.088,E2 -20114.088} C_VEL
LIN {X 0,Y 261.487,Z 194.703,A -85,B 0,C 180,E1 -20116.265,E2 -20116.265} C_VEL
LIN {X 0,Y 251.224,Z 310.134,A -85,B 0,C 180,E1 -20121.12,E2 -20121.12} C_VEL
LIN {X 0,Y 249.523,Z 327.21,A -85,B 0,C 180,E1 -20122.158,E2 -20122.158} C_VEL
LIN {X 0,Y 247.24,Z 345.49,A -85,B 0,C 180,E1 -20123.602,E2 -20123.602} C_VEL
LIN {X 0,Y 244.577,Z 363.516,A -85,B 0,C 180,E1 -20125.422,E2 -20125.422} C_VEL
LIN {X 0,Y 241.918,Z 379.499,A -85,B 0,C 180,E1 -20127.405,E2 -20127.405} C_VEL
LIN {X 0,Y 238.971,Z 395.206,A -85,B 0,C 180,E1 -20129.759,E2 -20129.759} C_VEL
LIN {X 0,Y 236.304,Z 409.343,A -85,B 0,C 180,E1 -20132.309,E2 -20132.309} C_VEL
LIN {X 0,Y 233.744,Z 422.386,A -85,B 0,C 180,E1 -20135.106,E2 -20135.106} C_VEL
LIN {X 0,Y 231.856,Z 432.775,A -85,B 0,C 180,E1 -20137.734,E2 -20137.734} C_VEL
LIN {X 0,Y 229.743,Z 444.399,A -85,B 0,C 180,E1 -20141.187,E2 -20141.187} C_VEL
LIN {X 0,Y 228.326,Z 453.436,A -85,B 0,C 180,E1 -20144.375,E2 -20144.375} C_VEL
LIN {X 0,Y 227.304,Z 460.921,A -85,B 0,C 180,E1 -20147.5,E2 -20147.5} C_VEL
LIN {X 0,Y 226.64,Z 468.057,A -85,B 0,C 180,E1 -20151.08,E2 -20151.08} C_VEL
LIN {X 0,Y 226.257,Z 473.894,A -85,B 0,C 180,E1 -20154.653,E2 -20154.653} C_VEL
LIN {X 0,Y 226.209,Z 478.518,A -85,B 0,C 180,E1 -20158.219,E2 -20158.219} C_VEL
LIN {X 0,Y 226.445,Z 481.999,A -85,B 0,C 180,E1 -20161.778,E2 -20161.778} C_VEL
LIN {X 0,Y 227.039,Z 484.546,A -85,B 0,C 180,E1 -20165.328,E2 -20165.328} C_VEL
LIN {X 0,Y 228.706,Z 486.48,A -85,B 0,C 180,E1 -20170.468,E2 -20170.468} C_VEL
LIN {X 0,Y 230.736,Z 486.67,A -85,B 0,C 180,E1 -20174.103,E2 -20174.103} C_VEL
LIN {X 0,Y 233.329,Z 486,A -85,B 0,C 180,E1 -20177.53,E2 -20177.53} C_VEL
LIN {X 0,Y 236.67,Z 484.432,A -85,B 0,C 180,E1 -20180.876,E2 -20180.876} C_VEL
LIN {X 0,Y 239.491,Z 482.826,A -85,B 0,C 180,E1 -20183.176,E2 -20183.176} C_VEL
LIN {X 0,Y 240.751,Z 481.921,A -85,B 0,C 180,E1 -20184.538,E2 -20184.538} C_VEL
LIN {X 0,Y 242.217,Z 479.518,A -85,B 0,C 180,E1 -20188.723,E2 -20188.723} C_VEL
LIN {X 0,Y 243.675,Z 478.265,A -85,B 0,C 180,E1 -20190.037,E2 -20190.037} C_VEL
LIN {X 0,Y 244.426,Z 477.738,A -85,B 0,C 180,E1 -20190.445,E2 -20190.445} C_VEL
LIN {X 0,Y 252.349,Z 472.398,A -85,B 0,C 180,E1 -20193.849,E2 -20193.849} C_VEL
LIN {X 0,Y 261.755,Z 465.5,A -85,B 0,C 180,E1 -20197.165,E2 -20197.165} C_VEL
LIN {X 0,Y 272.308,Z 457.23,A -85,B 0,C 180,E1 -20200.182,E2 -20200.182} C_VEL
LIN {X 0,Y 281.529,Z 449.571,A -85,B 0,C 180,E1 -20202.378,E2 -20202.378} C_VEL
LIN {X 0,Y 283.506,Z 448.027,A -85,B 0,C 180,E1 -20203.178,E2 -20203.178} C_VEL
LIN {X 0,Y 271.308,Z 460.03,A -85,B 0,C 180,E1 -20205.619,E2 -20205.619} C_VEL
LIN {X 0,Y 259.917,Z 470.98,A -85,B 0,C 180,E1 -20208.511,E2 -20208.511} C_VEL
LIN {X 0,Y 249.83,Z 480.687,A -85,B 0,C 180,E1 -20211.764,E2 -20211.764} C_VEL
LIN {X 0,Y 241.011,Z 489.216,A -85,B 0,C 180,E1 -20215.344,E2 -20215.344} C_VEL
LIN {X 0,Y 233.788,Z 496.442,A -85,B 0,C 180,E1 -20219.265,E2 -20219.265} C_VEL
LIN {X 0,Y 227.96,Z 502.403,A -85,B 0,C 180,E1 -20223.388,E2 -20223.388} C_VEL
LIN {X 0,Y 223.507,Z 507.287,A -85,B 0,C 180,E1 -20227.83,E2 -20227.83} C_VEL
LIN {X 0,Y 220.293,Z 511.348,A -85,B 0,C 180,E1 -20233.313,E2 -20233.313} C_VEL
LIN {X 0,Y 219.121,Z 512.963,A -85,B 0,C 180,E1 -20237.024,E2 -20237.024} C_VEL
LIN {X 0,Y 218.819,Z 513.753,A -85,B 0,C 180,E1 -20240.758,E2 -20240.758} C_VEL
LIN {X 0,Y 219.169,Z 513.519,A -85,B 0,C 180,E1 -20244.478,E2 -20244.478} C_VEL
LIN {X 0,Y 219.597,Z 512.261,A -85,B 0,C 180,E1 -20248.165,E2 -20248.165} C_VEL
LIN {X 0,Y 219.874,Z 511.179,A -85,B 0,C 180,E1 -20249.999,E2 -20249.999} C_VEL
LIN {X 0,Y 219.731,Z 508.041,A -85,B 0,C 180,E1 -20253.666,E2 -20253.666} C_VEL
LIN {X 0,Y 219.717,Z 504.302,A -85,B 0,C 180,E1 -20256.774,E2 -20256.774} C_VEL
LIN {X 0,Y 219.569,Z 499.162,A -85,B 0,C 180,E1 -20260.138,E2 -20260.138} C_VEL
LIN {X 0,Y 219.942,Z 492.02,A -85,B 0,C 180,E1 -20263.865,E2 -20263.865} C_VEL
LIN {X 0,Y 220.863,Z 483.166,A -85,B 0,C 180,E1 -20267.598,E2 -20267.598} C_VEL
LIN {X 0,Y 222.105,Z 473.863,A -85,B 0,C 180,E1 -20270.852,E2 -20270.852} C_VEL
LIN {X 0,Y 224.009,Z 462.963,A -85,B 0,C 180,E1 -20274.069,E2 -20274.069} C_VEL
LIN {X 0,Y 226.284,Z 451.103,A -85,B 0,C 180,E1 -20277.014,E2 -20277.014} C_VEL
LIN {X 0,Y 228.827,Z 438.334,A -85,B 0,C 180,E1 -20279.685,E2 -20279.685} C_VEL
LIN {X 0,Y 231.883,Z 423.423,A -85,B 0,C 180,E1 -20282.277,E2 -20282.277} C_VEL
LIN {X 0,Y 235.084,Z 407.023,A -85,B 0,C 180,E1 -20284.611,E2 -20284.611} C_VEL
LIN {X 0,Y 238.17,Z 390.064,A -85,B 0,C 180,E1 -20286.561,E2 -20286.561} C_VEL
LIN {X 0,Y 240.933,Z 373.42,A -85,B 0,C 180,E1 -20288.09,E2 -20288.09} C_VEL
LIN {X 0,Y 243.458,Z 355.664,A -85,B 0,C 180,E1 -20289.351,E2 -20289.351} C_VEL
LIN {X 0,Y 245.354,Z 337.22,A -85,B 0,C 180,E1 -20290.328,E2 -20290.328} C_VEL
LIN {X 0,Y 257.188,Z 211.33,A -85,B 0,C 180,E1 -20295.767,E2 -20295.767} C_VEL
LIN {X 0,Y 245.495,Z 183.789,A -85,B 0,C 180,E1 -20298.819,E2 -20298.819} C_VEL
LIN {X 0,Y 233.86,Z 158.194,A -85,B 0,C 180,E1 -20302.097,E2 -20302.097} C_VEL
LIN {X 0,Y 224.442,Z 138.87,A -85,B 0,C 180,E1 -20304.943,E2 -20304.943} C_VEL
LIN {X 0,Y 223.075,Z 135.864,A -85,B 0,C 180,E1 -20305.453,E2 -20305.453} C_VEL
LIN {X 0,Y 220.872,Z 129.285,A -85,B 0,C 180,E1 -20307.457,E2 -20307.457} C_VEL
LIN {X 0,Y 220.832,Z 129.291,A -85,B 0,C 180,E1 -20311.486,E2 -20311.486} C_VEL
LIN {X 0,Y 220.863,Z 129.29,A -85,B 0,C 180,E1 -20315.565,E2 -20315.565} C_VEL
LIN {X 0,Y 220.889,Z 129.282,A -85,B 0,C 180,E1 -20319.514,E2 -20319.514} C_VEL
LIN {X 0,Y 221.012,Z 129.263,A -85,B 0,C 180,E1 -20323.37,E2 -20323.37} C_VEL
LIN {X 0,Y 221.113,Z 129.249,A -85,B 0,C 180,E1 -20329.006,E2 -20329.006} C_VEL
LIN {X 0,Y 221.307,Z 129.229,A -85,B 0,C 180,E1 -20332.702,E2 -20332.702} C_VEL
LIN {X 0,Y 221.509,Z 129.206,A -85,B 0,C 180,E1 -20338.182,E2 -20338.182} C_VEL
LIN {X 0,Y 221.509,Z 129.204,A -85,B 0,C 180,E1 -20341.818,E2 -20341.818} C_VEL
LIN {X 0,Y 221.308,Z 129.228,A -85,B 0,C 180,E1 -20347.298,E2 -20347.298} C_VEL
LIN {X 0,Y 221.113,Z 129.252,A -85,B 0,C 180,E1 -20350.994,E2 -20350.994} C_VEL
LIN {X 0,Y 221.013,Z 129.264,A -85,B 0,C 180,E1 -20356.63,E2 -20356.63} C_VEL
LIN {X 0,Y 220.889,Z 129.281,A -85,B 0,C 180,E1 -20360.487,E2 -20360.487} C_VEL
LIN {X 0,Y 220.864,Z 129.278,A -85,B 0,C 180,E1 -20364.436,E2 -20364.436} C_VEL
LIN {X 0,Y 220.833,Z 129.288,A -85,B 0,C 180,E1 -20368.514,E2 -20368.514} C_VEL
LIN {X 0,Y 220.814,Z 129.288,A -85,B 0,C 180,E1 -20372.757,E2 -20372.757} C_VEL
LIN {X 0,Y 220.806,Z 129.288,A -85,B 0,C 180,E1 -20377.279,E2 -20377.279} C_VEL
LIN {X 0,Y 220.768,Z 129.296,A -85,B 0,C 180,E1 -20381.953,E2 -20381.953} C_VEL
LIN {X 0,Y 220.828,Z 129.284,A -85,B 0,C 180,E1 -20387.054,E2 -20387.054} C_VEL
LIN {X 0,Y 220.848,Z 129.288,A -85,B 0,C 180,E1 -20390.474,E2 -20390.474} C_VEL
LIN {X 0,Y 220.814,Z 129.288,A -85,B 0,C 180,E1 -20395.049,E2 -20395.049} C_VEL
LIN {X 0,Y 220.867,Z 129.282,A -85,B 0,C 180,E1 -20399.396,E2 -20399.396} C_VEL
LIN {X 0,Y 220.894,Z 129.279,A -85,B 0,C 180,E1 -20403.551,E2 -20403.551} C_VEL
LIN {X 0,Y 220.923,Z 129.274,A -85,B 0,C 180,E1 -20407.56,E2 -20407.56} C_VEL
LIN {X 0,Y 220.985,Z 129.271,A -85,B 0,C 180,E1 -20412.572,E2 -20412.572} C_VEL
LIN {X 0,Y 221.014,Z 129.265,A -85,B 0,C 180,E1 -20417.14,E2 -20417.14} C_VEL
LIN {X 0,Y 221.258,Z 129.231,A -85,B 0,C 180,E1 -20420.863,E2 -20420.863} C_VEL
LIN {X 0,Y 221.312,Z 129.229,A -85,B 0,C 180,E1 -20422.704,E2 -20422.704} C_VEL
LIN {X 0,Y 221.513,Z 129.205,A -85,B 0,C 180,E1 -20428.183,E2 -20428.183} C_VEL
LIN {X 0,Y 221.513,Z 129.199,A -85,B 0,C 180,E1 -20431.819,E2 -20431.819} C_VEL
LIN {X 0,Y 221.313,Z 129.23,A -85,B 0,C 180,E1 -20437.299,E2 -20437.299} C_VEL
LIN {X 0,Y 221.119,Z 129.247,A -85,B 0,C 180,E1 -20440.995,E2 -20440.995} C_VEL
LIN {X 0,Y 221.019,Z 129.264,A -85,B 0,C 180,E1 -20446.631,E2 -20446.631} C_VEL
LIN {X 0,Y 220.896,Z 129.281,A -85,B 0,C 180,E1 -20450.487,E2 -20450.487} C_VEL
LIN {X 0,Y 220.871,Z 129.284,A -85,B 0,C 180,E1 -20454.436,E2 -20454.436} C_VEL
LIN {X 0,Y 220.839,Z 129.289,A -85,B 0,C 180,E1 -20458.514,E2 -20458.514} C_VEL
LIN {X 0,Y 220.828,Z 129.291,A -85,B 0,C 180,E1 -20462.756,E2 -20462.756} C_VEL
LIN {X 0,Y 220.861,Z 129.287,A -85,B 0,C 180,E1 -20466.348,E2 -20466.348} C_VEL
LIN {X 0,Y 221.926,Z 132.232,A -85,B 0,C 180,E1 -20466.78,E2 -20466.78} C_VEL
LIN {X 0,Y 223.672,Z 135.282,A -85,B 0,C 180,E1 -20467.293,E2 -20467.293} C_VEL
LIN {X 0,Y 234.412,Z 155.139,A -85,B 0,C 180,E1 -20470.348,E2 -20470.348} C_VEL
LIN {X 0,Y 246.846,Z 179.657,A -85,B 0,C 180,E1 -20473.595,E2 -20473.595} C_VEL
LIN {X 0,Y 255.116,Z 196.814,A -85,B 0,C 180,E1 -20475.605,E2 -20475.605} C_VEL
LIN {X 0,Y 244.608,Z 310.461,A -85,B 0,C 180,E1 -20480.529,E2 -20480.529} C_VEL
LIN {X 0,Y 242.784,Z 328.13,A -85,B 0,C 180,E1 -20481.639,E2 -20481.639} C_VEL
LIN {X 0,Y 240.524,Z 345.702,A -85,B 0,C 180,E1 -20483.071,E2 -20483.071} C_VEL
LIN {X 0,Y 237.935,Z 362.883,A -85,B 0,C 180,E1 -20484.832,E2 -20484.832} C_VEL
LIN {X 0,Y 235.077,Z 379.683,A -85,B 0,C 180,E1 -20486.955,E2 -20486.955} C_VEL
LIN {X 0,Y 232.16,Z 394.854,A -85,B 0,C 180,E1 -20489.28,E2 -20489.28} C_VEL
LIN {X 0,Y 229.198,Z 410.197,A -85,B 0,C 180,E1 -20492.12,E2 -20492.12} C_VEL
LIN {X 0,Y 226.437,Z 424.125,A -85,B 0,C 180,E1 -20495.228,E2 -20495.228} C_VEL
LIN {X 0,Y 224.174,Z 435.972,A -85,B 0,C 180,E1 -20498.385,E2 -20498.385} C_VEL
LIN {X 0,Y 222.174,Z 447.406,A -85,B 0,C 180,E1 -20502.036,E2 -20502.036} C_VEL
LIN {X 0,Y 220.716,Z 456.958,A -85,B 0,C 180,E1 -20505.713,E2 -20505.713} C_VEL
LIN {X 0,Y 219.898,Z 463.991,A -85,B 0,C 180,E1 -20508.944,E2 -20508.944} C_VEL
LIN {X 0,Y 219.36,Z 470.728,A -85,B 0,C 180,E1 -20512.637,E2 -20512.637} C_VEL
LIN {X 0,Y 219.149,Z 476.13,A -85,B 0,C 180,E1 -20516.322,E2 -20516.322} C_VEL
LIN {X 0,Y 219.167,Z 480.381,A -85,B 0,C 180,E1 -20520,E2 -20520} C_VEL
LIN {X 0,Y 219.654,Z 483.612,A -85,B 0,C 180,E1 -20523.669,E2 -20523.669} C_VEL
LIN {X 0,Y 220.393,Z 485.806,A -85,B 0,C 180,E1 -20527.328,E2 -20527.328} C_VEL
LIN {X 0,Y 221.829,Z 487.144,A -85,B 0,C 180,E1 -20530.958,E2 -20530.958} C_VEL
LIN {X 0,Y 225.175,Z 487.437,A -85,B 0,C 180,E1 -20536.314,E2 -20536.314} C_VEL
LIN {X 0,Y 230.173,Z 485.793,A -85,B 0,C 180,E1 -20541.494,E2 -20541.494} C_VEL
LIN {X 0,Y 234.523,Z 483.667,A -85,B 0,C 180,E1 -20544.805,E2 -20544.805} C_VEL
LIN {X 0,Y 242.551,Z 478.966,A -85,B 0,C 180,E1 -20549.51,E2 -20549.51} C_VEL
LIN {X 0,Y 244.426,Z 477.738,A -85,B 0,C 180,E1 -20550.445,E2 -20550.445} C_VEL
LIN {X 0,Y 246.444,Z 476.295,A -85,B 0,C 180,E1 -20551.698,E2 -20551.698} C_VEL
LIN {X 0,Y 250.574,Z 472.728,A -85,B 0,C 180,E1 -20555.617,E2 -20555.617} C_VEL
LIN {X 0,Y 252.852,Z 471.12,A -85,B 0,C 180,E1 -20556.797,E2 -20556.797} C_VEL
LIN {X 0,Y 253.843,Z 470.474,A -85,B 0,C 180,E1 -20557.151,E2 -20557.151} C_VEL
LIN {X 0,Y 265.285,Z 462.56,A -85,B 0,C 180,E1 -20560.47,E2 -20560.47} C_VEL
LIN {X 0,Y 274.831,Z 455.465,A -85,B 0,C 180,E1 -20562.746,E2 -20562.746} C_VEL
LIN {X 0,Y 274.243,Z 456.072,A -85,B 0,C 180,E1 -20563.082,E2 -20563.082} C_VEL
LIN {X 0,Y 261.762,Z 467.176,A -85,B 0,C 180,E1 -20565.726,E2 -20565.726} C_VEL
LIN {X 0,Y 250.547,Z 477.045,A -85,B 0,C 180,E1 -20568.761,E2 -20568.761} C_VEL
LIN {X 0,Y 240.637,Z 485.661,A -85,B 0,C 180,E1 -20572.169,E2 -20572.169} C_VEL
LIN {X 0,Y 233.638,Z 491.809,A -85,B 0,C 180,E1 -20575.142,E2 -20575.142} C_VEL
LIN {X 0,Y 225.037,Z 499.557,A -85,B 0,C 180,E1 -20580.019,E2 -20580.019} C_VEL
LIN {X 0,Y 220.471,Z 503.771,A -85,B 0,C 180,E1 -20583.493,E2 -20583.493} C_VEL
LIN {X 0,Y 216.857,Z 507.221,A -85,B 0,C 180,E1 -20587.113,E2 -20587.113} C_VEL
LIN {X 0,Y 214.327,Z 509.931,A -85,B 0,C 180,E1 -20590.857,E2 -20590.857} C_VEL
LIN {X 0,Y 212.136,Z 512.411,A -85,B 0,C 180,E1 -20596.589,E2 -20596.589} C_VEL
LIN {X 0,Y 211.768,Z 512.952,A -85,B 0,C 180,E1 -20600.447,E2 -20600.447} C_VEL
LIN {X 0,Y 212.126,Z 512.575,A -85,B 0,C 180,E1 -20604.294,E2 -20604.294} C_VEL
LIN {X 0,Y 212.574,Z 511.163,A -85,B 0,C 180,E1 -20608.104,E2 -20608.104} C_VEL
LIN {X 0,Y 212.859,Z 510.016,A -85,B 0,C 180,E1 -20609.999,E2 -20609.999} C_VEL
LIN {X 0,Y 212.732,Z 506.632,A -85,B 0,C 180,E1 -20613.787,E2 -20613.787} C_VEL
LIN {X 0,Y 212.715,Z 502.912,A -85,B 0,C 180,E1 -20616.892,E2 -20616.892} C_VEL
LIN {X 0,Y 212.577,Z 497.366,A -85,B 0,C 180,E1 -20620.475,E2 -20620.475} C_VEL
LIN {X 0,Y 213.008,Z 489.979,A -85,B 0,C 180,E1 -20624.326,E2 -20624.326} C_VEL
LIN {X 0,Y 214.02,Z 480.889,A -85,B 0,C 180,E1 -20628.175,E2 -20628.175} C_VEL
LIN {X 0,Y 215.358,Z 471.296,A -85,B 0,C 180,E1 -20631.537,E2 -20631.537} C_VEL
LIN {X 0,Y 217.41,Z 460.01,A -85,B 0,C 180,E1 -20634.848,E2 -20634.848} C_VEL
LIN {X 0,Y 220.068,Z 446.72,A -85,B 0,C 180,E1 -20638.101,E2 -20638.101} C_VEL
LIN {X 0,Y 222.794,Z 433.292,A -85,B 0,C 180,E1 -20640.836,E2 -20640.836} C_VEL
LIN {X 0,Y 225.77,Z 418.953,A -85,B 0,C 180,E1 -20643.272,E2 -20643.272} C_VEL
LIN {X 0,Y 228.85,Z 403.639,A -85,B 0,C 180,E1 -20645.425,E2 -20645.425} C_VEL
LIN {X 0,Y 231.826,Z 387.076,A -85,B 0,C 180,E1 -20647.322,E2 -20647.322} C_VEL
LIN {X 0,Y 234.804,Z 369.094,A -85,B 0,C 180,E1 -20648.942,E2 -20648.942} C_VEL
LIN {X 0,Y 237.196,Z 352.054,A -85,B 0,C 180,E1 -20650.122,E2 -20650.122} C_VEL
LIN {X 0,Y 239.417,Z 329.902,A -85,B 0,C 180,E1 -20651.265,E2 -20651.265} C_VEL
LIN {X 0,Y 250.797,Z 213.253,A -85,B 0,C 180,E1 -20656.45,E2 -20656.45} C_VEL
LIN {X 0,Y 239.969,Z 187.569,A -85,B 0,C 180,E1 -20659.377,E2 -20659.377} C_VEL
LIN {X 0,Y 228.331,Z 161.761,A -85,B 0,C 180,E1 -20662.77,E2 -20662.77} C_VEL
LIN {X 0,Y 217.88,Z 140.074,A -85,B 0,C 180,E1 -20666.059,E2 -20666.059} C_VEL
LIN {X 0,Y 215.559,Z 135.306,A -85,B 0,C 180,E1 -20666.9,E2 -20666.9} C_VEL
LIN {X 0,Y 213.789,Z 130.166,A -85,B 0,C 180,E1 -20668.552,E2 -20668.552} C_VEL
LIN {X 0,Y 213.822,Z 130.167,A -85,B 0,C 180,E1 -20672.603,E2 -20672.603} C_VEL
LIN {X 0,Y 213.848,Z 130.162,A -85,B 0,C 180,E1 -20676.953,E2 -20676.953} C_VEL
LIN {X 0,Y 213.94,Z 130.144,A -85,B 0,C 180,E1 -20682.804,E2 -20682.804} C_VEL
LIN {X 0,Y 213.977,Z 130.138,A -85,B 0,C 180,E1 -20686.708,E2 -20686.708} C_VEL
LIN {X 0,Y 214.192,Z 130.117,A -85,B 0,C 180,E1 -20690.558,E2 -20690.558} C_VEL
LIN {X 0,Y 214.244,Z 130.109,A -85,B 0,C 180,E1 -20692.46,E2 -20692.46} C_VEL
LIN {X 0,Y 214.442,Z 130.086,A -85,B 0,C 180,E1 -20698.122,E2 -20698.122} C_VEL
LIN {X 0,Y 214.551,Z 130.071,A -85,B 0,C 180,E1 -20700,E2 -20700} C_VEL
LIN {X 0,Y 214.443,Z 130.084,A -85,B 0,C 180,E1 -20701.878,E2 -20701.878} C_VEL
LIN {X 0,Y 214.244,Z 130.109,A -85,B 0,C 180,E1 -20707.54,E2 -20707.54} C_VEL
LIN {X 0,Y 214.044,Z 130.131,A -85,B 0,C 180,E1 -20711.362,E2 -20711.362} C_VEL
LIN {X 0,Y 213.93,Z 130.151,A -85,B 0,C 180,E1 -20715.237,E2 -20715.237} C_VEL
LIN {X 0,Y 213.836,Z 130.159,A -85,B 0,C 180,E1 -20719.188,E2 -20719.188} C_VEL
LIN {X 0,Y 213.844,Z 130.155,A -85,B 0,C 180,E1 -20723.228,E2 -20723.228} C_VEL
LIN {X 0,Y 213.825,Z 130.163,A -85,B 0,C 180,E1 -20727.451,E2 -20727.451} C_VEL
LIN {X 0,Y 213.773,Z 130.163,A -85,B 0,C 180,E1 -20731.737,E2 -20731.737} C_VEL
LIN {X 0,Y 213.74,Z 130.171,A -85,B 0,C 180,E1 -20736.289,E2 -20736.289} C_VEL
LIN {X 0,Y 213.709,Z 130.177,A -85,B 0,C 180,E1 -20741.126,E2 -20741.126} C_VEL
LIN {X 0,Y 213.774,Z 130.161,A -85,B 0,C 180,E1 -20746.341,E2 -20746.341} C_VEL
LIN {X 0,Y 213.777,Z 130.166,A -85,B 0,C 180,E1 -20751.346,E2 -20751.346} C_VEL
LIN {X 0,Y 213.767,Z 130.166,A -85,B 0,C 180,E1 -20756.021,E2 -20756.021} C_VEL
LIN {X 0,Y 213.779,Z 130.164,A -85,B 0,C 180,E1 -20760.455,E2 -20760.455} C_VEL
LIN {X 0,Y 213.804,Z 130.166,A -85,B 0,C 180,E1 -20764.704,E2 -20764.704} C_VEL
LIN {X 0,Y 213.84,Z 130.155,A -85,B 0,C 180,E1 -20768.808,E2 -20768.808} C_VEL
LIN {X 0,Y 213.944,Z 130.147,A -85,B 0,C 180,E1 -20772.805,E2 -20772.805} C_VEL
LIN {X 0,Y 213.955,Z 130.146,A -85,B 0,C 180,E1 -20776.708,E2 -20776.708} C_VEL
LIN {X 0,Y 214.197,Z 130.111,A -85,B 0,C 180,E1 -20780.559,E2 -20780.559} C_VEL
LIN {X 0,Y 214.249,Z 130.109,A -85,B 0,C 180,E1 -20782.462,E2 -20782.462} C_VEL
LIN {X 0,Y 214.447,Z 130.084,A -85,B 0,C 180,E1 -20788.123,E2 -20788.123} C_VEL
LIN {X 0,Y 214.551,Z 130.073,A -85,B 0,C 180,E1 -20790.001,E2 -20790.001} C_VEL
LIN {X 0,Y 214.447,Z 130.078,A -85,B 0,C 180,E1 -20791.879,E2 -20791.879} C_VEL
LIN {X 0,Y 214.25,Z 130.111,A -85,B 0,C 180,E1 -20797.541,E2 -20797.541} C_VEL
LIN {X 0,Y 214.05,Z 130.126,A -85,B 0,C 180,E1 -20801.363,E2 -20801.363} C_VEL
LIN {X 0,Y 213.937,Z 130.151,A -85,B 0,C 180,E1 -20805.238,E2 -20805.238} C_VEL
LIN {X 0,Y 213.843,Z 130.155,A -85,B 0,C 180,E1 -20809.188,E2 -20809.188} C_VEL
LIN {X 0,Y 213.85,Z 130.153,A -85,B 0,C 180,E1 -20813.228,E2 -20813.228} C_VEL
LIN {X 0,Y 213.832,Z 130.158,A -85,B 0,C 180,E1 -20817.451,E2 -20817.451} C_VEL
LIN {X 0,Y 213.783,Z 130.165,A -85,B 0,C 180,E1 -20821.736,E2 -20821.736} C_VEL
LIN {X 0,Y 213.777,Z 130.192,A -85,B 0,C 180,E1 -20825.122,E2 -20825.122} C_VEL
LIN {X 0,Y 214.964,Z 133.287,A -85,B 0,C 180,E1 -20825.567,E2 -20825.567} C_VEL
LIN {X 0,Y 216.089,Z 135.067,A -85,B 0,C 180,E1 -20825.905,E2 -20825.905} C_VEL
LIN {X 0,Y 228.243,Z 157.608,A -85,B 0,C 180,E1 -20829.53,E2 -20829.53} C_VEL
LIN {X 0,Y 239.652,Z 180.127,A -85,B 0,C 180,E1 -20832.63,E2 -20832.63} C_VEL
LIN {X 0,Y 248.637,Z 198.854,A -85,B 0,C 180,E1 -20834.902,E2 -20834.902} C_VEL
LIN {X 0,Y 237.967,Z 311.254,A -85,B 0,C 180,E1 -20839.944,E2 -20839.944} C_VEL
LIN {X 0,Y 236.015,Z 329.372,A -85,B 0,C 180,E1 -20841.128,E2 -20841.128} C_VEL
LIN {X 0,Y 233.49,Z 347.943,A -85,B 0,C 180,E1 -20842.717,E2 -20842.717} C_VEL
LIN {X 0,Y 231.028,Z 363.898,A -85,B 0,C 180,E1 -20844.423,E2 -20844.423} C_VEL
LIN {X 0,Y 228.101,Z 380.429,A -85,B 0,C 180,E1 -20846.582,E2 -20846.582} C_VEL
LIN {X 0,Y 224.867,Z 396.947,A -85,B 0,C 180,E1 -20849.217,E2 -20849.217} C_VEL
LIN {X 0,Y 221.921,Z 411.688,A -85,B 0,C 180,E1 -20852.076,E2 -20852.076} C_VEL
LIN {X 0,Y 219.481,Z 423.925,A -85,B 0,C 180,E1 -20854.895,E2 -20854.895} C_VEL
LIN {X 0,Y 217.482,Z 434.238,A -85,B 0,C 180,E1 -20857.684,E2 -20857.684} C_VEL
LIN {X 0,Y 215.385,Z 445.726,A -85,B 0,C 180,E1 -20861.328,E2 -20861.328} C_VEL
LIN {X 0,Y 213.934,Z 454.802,A -85,B 0,C 180,E1 -20864.763,E2 -20864.763} C_VEL
LIN {X 0,Y 212.865,Z 463.265,A -85,B 0,C 180,E1 -20868.574,E2 -20868.574} C_VEL
LIN {X 0,Y 212.302,Z 470.197,A -85,B 0,C 180,E1 -20872.391,E2 -20872.391} C_VEL
LIN {X 0,Y 212.06,Z 475.836,A -85,B 0,C 180,E1 -20876.199,E2 -20876.199} C_VEL
LIN {X 0,Y 212.085,Z 480.351,A -85,B 0,C 180,E1 -20880,E2 -20880} C_VEL
LIN {X 0,Y 212.584,Z 483.719,A -85,B 0,C 180,E1 -20883.791,E2 -20883.791} C_VEL
LIN {X 0,Y 213.36,Z 486.199,A -85,B 0,C 180,E1 -20887.571,E2 -20887.571} C_VEL
LIN {X 0,Y 214.871,Z 487.684,A -85,B 0,C 180,E1 -20891.317,E2 -20891.317} C_VEL
LIN {X 0,Y 217.058,Z 488.374,A -85,B 0,C 180,E1 -20895.012,E2 -20895.012} C_VEL
LIN {X 0,Y 221.752,Z 487.731,A -85,B 0,C 180,E1 -20900.403,E2 -20900.403} C_VEL
LIN {X 0,Y 225.837,Z 486.284,A -85,B 0,C 180,E1 -20903.863,E2 -20903.863} C_VEL
LIN {X 0,Y 230.908,Z 484.064,A -85,B 0,C 180,E1 -20907.164,E2 -20907.164} C_VEL
LIN {X 0,Y 239.868,Z 479.211,A -85,B 0,C 180,E1 -20911.829,E2 -20911.829} C_VEL
LIN {X 0,Y 248.766,Z 473.81,A -85,B 0,C 180,E1 -20915.391,E2 -20915.391} C_VEL
LIN {X 0,Y 253.843,Z 470.474,A -85,B 0,C 180,E1 -20917.151,E2 -20917.151} C_VEL
LIN {X 0,Y 255.551,Z 469.357,A -85,B 0,C 180,E1 -20917.926,E2 -20917.926} C_VEL
LIN {X 0,Y 259.019,Z 466.997,A -85,B 0,C 180,E1 -20920.785,E2 -20920.785} C_VEL
LIN {X 0,Y 260.984,Z 465.713,A -85,B 0,C 180,E1 -20921.49,E2 -20921.49} C_VEL
LIN {X 0,Y 265.739,Z 462.605,A -85,B 0,C 180,E1 -20922.621,E2 -20922.621} C_VEL
LIN {X 0,Y 264.546,Z 463.675,A -85,B 0,C 180,E1 -20923.064,E2 -20923.064} C_VEL
LIN {X 0,Y 254.588,Z 471.659,A -85,B 0,C 180,E1 -20925.255,E2 -20925.255} C_VEL
LIN {X 0,Y 243.28,Z 480.68,A -85,B 0,C 180,E1 -20928.36,E2 -20928.36} C_VEL
LIN {X 0,Y 231.354,Z 490.03,A -85,B 0,C 180,E1 -20932.586,E2 -20932.586} C_VEL
LIN {X 0,Y 221.707,Z 497.772,A -85,B 0,C 180,E1 -20937.391,E2 -20937.391} C_VEL
LIN {X 0,Y 214.723,Z 503.405,A -85,B 0,C 180,E1 -20942.094,E2 -20942.094} C_VEL
LIN {X 0,Y 210.253,Z 507.192,A -85,B 0,C 180,E1 -20946.351,E2 -20946.351} C_VEL
LIN {X 0,Y 206.42,Z 510.668,A -85,B 0,C 180,E1 -20952.423,E2 -20952.423} C_VEL
LIN {X 0,Y 204.816,Z 512.076,A -85,B 0,C 180,E1 -20958.118,E2 -20958.118} C_VEL
LIN {X 0,Y 205.008,Z 511.672,A -85,B 0,C 180,E1 -20963.803,E2 -20963.803} C_VEL
LIN {X 0,Y 205.33,Z 510.92,A -85,B 0,C 180,E1 -20966.073,E2 -20966.073} C_VEL
LIN {X 0,Y 205.857,Z 508.757,A -85,B 0,C 180,E1 -20969.999,E2 -20969.999} C_VEL
LIN {X 0,Y 205.771,Z 507.167,A -85,B 0,C 180,E1 -20971.956,E2 -20971.956} C_VEL
LIN {X 0,Y 205.736,Z 502.905,A -85,B 0,C 180,E1 -20975.881,E2 -20975.881} C_VEL
LIN {X 0,Y 205.591,Z 498.782,A -85,B 0,C 180,E1 -20978.848,E2 -20978.848} C_VEL
LIN {X 0,Y 205.747,Z 491.875,A -85,B 0,C 180,E1 -20982.827,E2 -20982.827} C_VEL
LIN {X 0,Y 206.413,Z 484.536,A -85,B 0,C 180,E1 -20986.312,E2 -20986.312} C_VEL
LIN {X 0,Y 207.562,Z 475.81,A -85,B 0,C 180,E1 -20989.79,E2 -20989.79} C_VEL
LIN {X 0,Y 209.254,Z 465.407,A -85,B 0,C 180,E1 -20993.242,E2 -20993.242} C_VEL
LIN {X 0,Y 211.598,Z 453.204,A -85,B 0,C 180,E1 -20996.638,E2 -20996.638} C_VEL
LIN {X 0,Y 214.102,Z 440.964,A -85,B 0,C 180,E1 -20999.496,E2 -20999.496} C_VEL
LIN {X 0,Y 217.109,Z 427.018,A -85,B 0,C 180,E1 -21002.228,E2 -21002.228} C_VEL
LIN {X 0,Y 220.328,Z 411.32,A -85,B 0,C 180,E1 -21004.761,E2 -21004.761} C_VEL
LIN {X 0,Y 223.627,Z 394.643,A -85,B 0,C 180,E1 -21006.943,E2 -21006.943} C_VEL
LIN {X 0,Y 226.708,Z 377.338,A -85,B 0,C 180,E1 -21008.755,E2 -21008.755} C_VEL
LIN {X 0,Y 229.477,Z 359.999,A -85,B 0,C 180,E1 -21010.169,E2 -21010.169} C_VEL
LIN {X 0,Y 231.63,Z 341.995,A -85,B 0,C 180,E1 -21011.293,E2 -21011.293} C_VEL
LIN {X 0,Y 244.435,Z 215.16,A -85,B 0,C 180,E1 -21017.161,E2 -21017.161} C_VEL
LIN {X 0,Y 234.026,Z 190.398,A -85,B 0,C 180,E1 -21020.066,E2 -21020.066} C_VEL
LIN {X 0,Y 222.649,Z 164.977,A -85,B 0,C 180,E1 -21023.501,E2 -21023.501} C_VEL
LIN {X 0,Y 212.389,Z 143.678,A -85,B 0,C 180,E1 -21026.837,E2 -21026.837} C_VEL
LIN {X 0,Y 208.007,Z 134.848,A -85,B 0,C 180,E1 -21028.395,E2 -21028.395} C_VEL
LIN {X 0,Y 206.731,Z 131.049,A -85,B 0,C 180,E1 -21029.694,E2 -21029.694} C_VEL
LIN {X 0,Y 206.729,Z 131.049,A -85,B 0,C 180,E1 -21033.772,E2 -21033.772} C_VEL
LIN {X 0,Y 206.754,Z 131.048,A -85,B 0,C 180,E1 -21038.043,E2 -21038.043} C_VEL
LIN {X 0,Y 206.869,Z 131.027,A -85,B 0,C 180,E1 -21042.196,E2 -21042.196} C_VEL
LIN {X 0,Y 206.91,Z 131.02,A -85,B 0,C 180,E1 -21046.246,E2 -21046.246} C_VEL
LIN {X 0,Y 207.129,Z 130.998,A -85,B 0,C 180,E1 -21050.233,E2 -21050.233} C_VEL
LIN {X 0,Y 207.185,Z 130.989,A -85,B 0,C 180,E1 -21052.202,E2 -21052.202} C_VEL
LIN {X 0,Y 207.379,Z 130.966,A -85,B 0,C 180,E1 -21058.058,E2 -21058.058} C_VEL
LIN {X 0,Y 207.515,Z 130.948,A -85,B 0,C 180,E1 -21060,E2 -21060} C_VEL
LIN {X 0,Y 207.084,Z 131.002,A -85,B 0,C 180,E1 -21063.892,E2 -21063.892} C_VEL
LIN {X 0,Y 207.185,Z 130.99,A -85,B 0,C 180,E1 -21067.798,E2 -21067.798} C_VEL
LIN {X 0,Y 206.98,Z 131.011,A -85,B 0,C 180,E1 -21071.755,E2 -21071.755} C_VEL
LIN {X 0,Y 206.864,Z 131.027,A -85,B 0,C 180,E1 -21075.771,E2 -21075.771} C_VEL
LIN {X 0,Y 206.781,Z 131.039,A -85,B 0,C 180,E1 -21079.87,E2 -21079.87} C_VEL
LIN {X 0,Y 206.76,Z 131.034,A -85,B 0,C 180,E1 -21084.073,E2 -21084.073} C_VEL
LIN {X 0,Y 206.741,Z 131.044,A -85,B 0,C 180,E1 -21088.419,E2 -21088.419} C_VEL
LIN {X 0,Y 206.699,Z 131.047,A -85,B 0,C 180,E1 -21092.958,E2 -21092.958} C_VEL
LIN {X 0,Y 206.676,Z 131.046,A -85,B 0,C 180,E1 -21097.741,E2 -21097.741} C_VEL
LIN {X 0,Y 206.639,Z 131.056,A -85,B 0,C 180,E1 -21101.564,E2 -21101.564} C_VEL
LIN {X 0,Y 206.675,Z 131.045,A -85,B 0,C 180,E1 -21105.57,E2 -21105.57} C_VEL
LIN {X 0,Y 206.701,Z 131.048,A -85,B 0,C 180,E1 -21109.76,E2 -21109.76} C_VEL
LIN {X 0,Y 206.722,Z 131.045,A -85,B 0,C 180,E1 -21112.271,E2 -21112.271} C_VEL
LIN {X 0,Y 206.708,Z 131.049,A -85,B 0,C 180,E1 -21117.046,E2 -21117.046} C_VEL
LIN {X 0,Y 206.765,Z 131.033,A -85,B 0,C 180,E1 -21122.098,E2 -21122.098} C_VEL
LIN {X 0,Y 206.792,Z 131.037,A -85,B 0,C 180,E1 -21126.58,E2 -21126.58} C_VEL
LIN {X 0,Y 206.878,Z 131.029,A -85,B 0,C 180,E1 -21132.198,E2 -21132.198} C_VEL
LIN {X 0,Y 206.897,Z 131.021,A -85,B 0,C 180,E1 -21136.246,E2 -21136.246} C_VEL
LIN {X 0,Y 207.133,Z 130.993,A -85,B 0,C 180,E1 -21140.234,E2 -21140.234} C_VEL
LIN {X 0,Y 207.189,Z 130.986,A -85,B 0,C 180,E1 -21142.203,E2 -21142.203} C_VEL
LIN {X 0,Y 207.383,Z 130.963,A -85,B 0,C 180,E1 -21148.059,E2 -21148.059} C_VEL
LIN {X 0,Y 207.516,Z 130.949,A -85,B 0,C 180,E1 -21150.001,E2 -21150.001} C_VEL
LIN {X 0,Y 207.383,Z 130.956,A -85,B 0,C 180,E1 -21151.943,E2 -21151.943} C_VEL
LIN {X 0,Y 207.191,Z 130.992,A -85,B 0,C 180,E1 -21157.799,E2 -21157.799} C_VEL
LIN {X 0,Y 206.986,Z 131.005,A -85,B 0,C 180,E1 -21161.756,E2 -21161.756} C_VEL
LIN {X 0,Y 206.87,Z 131.031,A -85,B 0,C 180,E1 -21165.772,E2 -21165.772} C_VEL
LIN {X 0,Y 206.787,Z 131.038,A -85,B 0,C 180,E1 -21169.87,E2 -21169.87} C_VEL
LIN {X 0,Y 206.767,Z 131.037,A -85,B 0,C 180,E1 -21174.073,E2 -21174.073} C_VEL
LIN {X 0,Y 206.747,Z 131.042,A -85,B 0,C 180,E1 -21178.42,E2 -21178.42} C_VEL
LIN {X 0,Y 206.713,Z 131.051,A -85,B 0,C 180,E1 -21182.957,E2 -21182.957} C_VEL
LIN {X 0,Y 206.734,Z 131.047,A -85,B 0,C 180,E1 -21183.754,E2 -21183.754} C_VEL
LIN {X 0,Y 207.766,Z 133.941,A -85,B 0,C 180,E1 -21184.221,E2 -21184.221} C_VEL
LIN {X 0,Y 209.071,Z 136.019,A -85,B 0,C 180,E1 -21184.637,E2 -21184.637} C_VEL
LIN {X 0,Y 218.336,Z 152.931,A -85,B 0,C 180,E1 -21187.56,E2 -21187.56} C_VEL
LIN {X 0,Y 229.985,Z 175.522,A -85,B 0,C 180,E1 -21190.939,E2 -21190.939} C_VEL
LIN {X 0,Y 241.995,Z 200.32,A -85,B 0,C 180,E1 -21194.125,E2 -21194.125} C_VEL
LIN {X 0,Y 242.255,Z 200.918,A -85,B 0,C 180,E1 -21194.194,E2 -21194.194} C_VEL
LIN {X 0,Y 231.291,Z 312.12,A -85,B 0,C 180,E1 -21199.352,E2 -21199.352} C_VEL
LIN {X 0,Y 229.36,Z 329.518,A -85,B 0,C 180,E1 -21200.519,E2 -21200.519} C_VEL
LIN {X 0,Y 226.801,Z 347.905,A -85,B 0,C 180,E1 -21202.125,E2 -21202.125} C_VEL
LIN {X 0,Y 224.058,Z 365.116,A -85,B 0,C 180,E1 -21204.031,E2 -21204.031} C_VEL
LIN {X 0,Y 221.101,Z 381.177,A -85,B 0,C 180,E1 -21206.202,E2 -21206.202} C_VEL
LIN {X 0,Y 218.085,Z 396.402,A -85,B 0,C 180,E1 -21208.692,E2 -21208.692} C_VEL
LIN {X 0,Y 214.98,Z 411.684,A -85,B 0,C 180,E1 -21211.716,E2 -21211.716} C_VEL
LIN {X 0,Y 212.174,Z 425.496,A -85,B 0,C 180,E1 -21215.018,E2 -21215.018} C_VEL
LIN {X 0,Y 209.822,Z 437.283,A -85,B 0,C 180,E1 -21218.38,E2 -21218.38} C_VEL
LIN {X 0,Y 207.869,Z 448.716,A -85,B 0,C 180,E1 -21222.284,E2 -21222.284} C_VEL
LIN {X 0,Y 206.323,Z 458.212,A -85,B 0,C 180,E1 -21226.205,E2 -21226.205} C_VEL
LIN {X 0,Y 205.497,Z 466.146,A -85,B 0,C 180,E1 -21230.154,E2 -21230.154} C_VEL
LIN {X 0,Y 205.032,Z 472.681,A -85,B 0,C 180,E1 -21234.097,E2 -21234.097} C_VEL
LIN {X 0,Y 204.985,Z 478.003,A -85,B 0,C 180,E1 -21238.035,E2 -21238.035} C_VEL
LIN {X 0,Y 205.205,Z 482.109,A -85,B 0,C 180,E1 -21241.962,E2 -21241.962} C_VEL
LIN {X 0,Y 205.893,Z 485.289,A -85,B 0,C 180,E1 -21245.877,E2 -21245.877} C_VEL
LIN {X 0,Y 207.448,Z 487.879,A -85,B 0,C 180,E1 -21250.738,E2 -21250.738} C_VEL
LIN {X 0,Y 210.23,Z 489.088,A -85,B 0,C 180,E1 -21255.512,E2 -21255.512} C_VEL
LIN {X 0,Y 213.323,Z 489.165,A -85,B 0,C 180,E1 -21259.235,E2 -21259.235} C_VEL
LIN {X 0,Y 219.488,Z 487.715,A -85,B 0,C 180,E1 -21264.598,E2 -21264.598} C_VEL
LIN {X 0,Y 224.805,Z 485.723,A -85,B 0,C 180,E1 -21267.965,E2 -21267.965} C_VEL
LIN {X 0,Y 230.836,Z 483.065,A -85,B 0,C 180,E1 -21271.17,E2 -21271.17} C_VEL
LIN {X 0,Y 241.477,Z 477.527,A -85,B 0,C 180,E1 -21275.597,E2 -21275.597} C_VEL
LIN {X 0,Y 251.6,Z 471.639,A -85,B 0,C 180,E1 -21278.939,E2 -21278.939} C_VEL
LIN {X 0,Y 260.984,Z 465.713,A -85,B 0,C 180,E1 -21281.49,E2 -21281.49} C_VEL
LIN {X 0,Y 261.369,Z 465.516,A -85,B 0,C 180,E1 -21281.776,E2 -21281.776} C_VEL
LIN {X 0,Y 260.697,Z 466.145,A -85,B 0,C 180,E1 -21282.297,E2 -21282.297} C_VEL
LIN {X 0,Y 258.598,Z 467.801,A -85,B 0,C 180,E1 -21282.878,E2 -21282.878} C_VEL
LIN {X 0,Y 249.105,Z 474.583,A -85,B 0,C 180,E1 -21284.367,E2 -21284.367} C_VEL
LIN {X 0,Y 248.005,Z 475.339,A -85,B 0,C 180,E1 -21284.615,E2 -21284.615} C_VEL
LIN {X 0,Y 236.006,Z 483.963,A -85,B 0,C 180,E1 -21287.93,E2 -21287.93} C_VEL
LIN {X 0,Y 224.019,Z 492.445,A -85,B 0,C 180,E1 -21292.282,E2 -21292.282} C_VEL
LIN {X 0,Y 214.249,Z 499.429,A -85,B 0,C 180,E1 -21297.23,E2 -21297.23} C_VEL
LIN {X 0,Y 207.716,Z 504.128,A -85,B 0,C 180,E1 -21301.725,E2 -21301.725} C_VEL
LIN {X 0,Y 202.081,Z 508.264,A -85,B 0,C 180,E1 -21307.506,E2 -21307.506} C_VEL
LIN {X 0,Y 198.816,Z 510.691,A -85,B 0,C 180,E1 -21313.572,E2 -21313.572} C_VEL
LIN {X 0,Y 197.68,Z 511.271,A -85,B 0,C 180,E1 -21319.759,E2 -21319.759} C_VEL
LIN {X 0,Y 198.037,Z 510.514,A -85,B 0,C 180,E1 -21323.887,E2 -21323.887} C_VEL
LIN {X 0,Y 198.323,Z 509.814,A -85,B 0,C 180,E1 -21325.934,E2 -21325.934} C_VEL
LIN {X 0,Y 198.868,Z 507.417,A -85,B 0,C 180,E1 -21329.999,E2 -21329.999} C_VEL
LIN {X 0,Y 198.747,Z 503.696,A -85,B 0,C 180,E1 -21334.054,E2 -21334.054} C_VEL
LIN {X 0,Y 198.697,Z 499.777,A -85,B 0,C 180,E1 -21337.22,E2 -21337.22} C_VEL
LIN {X 0,Y 198.602,Z 493.59,A -85,B 0,C 180,E1 -21341.222,E2 -21341.222} C_VEL
LIN {X 0,Y 199.194,Z 485.659,A -85,B 0,C 180,E1 -21345.343,E2 -21345.343} C_VEL
LIN {X 0,Y 200.373,Z 475.879,A -85,B 0,C 180,E1 -21349.461,E2 -21349.461} C_VEL
LIN {X 0,Y 202.032,Z 465.638,A -85,B 0,C 180,E1 -21353.037,E2 -21353.037} C_VEL
LIN {X 0,Y 204.416,Z 453.325,A -85,B 0,C 180,E1 -21356.633,E2 -21356.633} C_VEL
LIN {X 0,Y 207.088,Z 440.476,A -85,B 0,C 180,E1 -21359.756,E2 -21359.756} C_VEL
LIN {X 0,Y 210.385,Z 425.471,A -85,B 0,C 180,E1 -21362.77,E2 -21362.77} C_VEL
LIN {X 0,Y 213.754,Z 409.379,A -85,B 0,C 180,E1 -21365.413,E2 -21365.413} C_VEL
LIN {X 0,Y 216.797,Z 394.334,A -85,B 0,C 180,E1 -21367.431,E2 -21367.431} C_VEL
LIN {X 0,Y 219.904,Z 377.282,A -85,B 0,C 180,E1 -21369.285,E2 -21369.285} C_VEL
LIN {X 0,Y 222.729,Z 360.076,A -85,B 0,C 180,E1 -21370.744,E2 -21370.744} C_VEL
LIN {X 0,Y 224.953,Z 342.319,A -85,B 0,C 180,E1 -21371.896,E2 -21371.896} C_VEL
LIN {X 0,Y 238.008,Z 216.905,A -85,B 0,C 180,E1 -21377.904,E2 -21377.904} C_VEL
LIN {X 0,Y 228.063,Z 193.183,A -85,B 0,C 180,E1 -21380.787,E2 -21380.787} C_VEL
LIN {X 0,Y 217.284,Z 168.88,A -85,B 0,C 180,E1 -21384.149,E2 -21384.149} C_VEL
LIN {X 0,Y 207.432,Z 148.19,A -85,B 0,C 180,E1 -21387.47,E2 -21387.47} C_VEL
LIN {X 0,Y 200.428,Z 134.288,A -85,B 0,C 180,E1 -21390.022,E2 -21390.022} C_VEL
LIN {X 0,Y 199.701,Z 131.923,A -85,B 0,C 180,E1 -21390.849,E2 -21390.849} C_VEL
LIN {X 0,Y 199.733,Z 131.92,A -85,B 0,C 180,E1 -21396.182,E2 -21396.182} C_VEL
LIN {X 0,Y 199.793,Z 131.911,A -85,B 0,C 180,E1 -21401.757,E2 -21401.757} C_VEL
LIN {X 0,Y 199.844,Z 131.903,A -85,B 0,C 180,E1 -21405.749,E2 -21405.749} C_VEL
LIN {X 0,Y 200.071,Z 131.873,A -85,B 0,C 180,E1 -21409.885,E2 -21409.885} C_VEL
LIN {X 0,Y 200.128,Z 131.87,A -85,B 0,C 180,E1 -21411.925,E2 -21411.925} C_VEL
LIN {X 0,Y 200.319,Z 131.846,A -85,B 0,C 180,E1 -21417.99,E2 -21417.99} C_VEL
LIN {X 0,Y 200.479,Z 131.824,A -85,B 0,C 180,E1 -21420,E2 -21420} C_VEL
LIN {X 0,Y 200.03,Z 131.88,A -85,B 0,C 180,E1 -21424.03,E2 -21424.03} C_VEL
LIN {X 0,Y 200.129,Z 131.868,A -85,B 0,C 180,E1 -21428.075,E2 -21428.075} C_VEL
LIN {X 0,Y 199.911,Z 131.892,A -85,B 0,C 180,E1 -21432.177,E2 -21432.177} C_VEL
LIN {X 0,Y 199.801,Z 131.906,A -85,B 0,C 180,E1 -21436.344,E2 -21436.344} C_VEL
LIN {X 0,Y 199.697,Z 131.921,A -85,B 0,C 180,E1 -21440.606,E2 -21440.606} C_VEL
LIN {X 0,Y 199.67,Z 131.919,A -85,B 0,C 180,E1 -21444.985,E2 -21444.985} C_VEL
LIN {X 0,Y 199.671,Z 131.921,A -85,B 0,C 180,E1 -21449.523,E2 -21449.523} C_VEL
LIN {X 0,Y 199.674,Z 131.919,A -85,B 0,C 180,E1 -21452.359,E2 -21452.359} C_VEL
LIN {X 0,Y 199.619,Z 131.93,A -85,B 0,C 180,E1 -21456.764,E2 -21456.764} C_VEL
LIN {X 0,Y 199.605,Z 131.927,A -85,B 0,C 180,E1 -21459.329,E2 -21459.329} C_VEL
LIN {X 0,Y 199.572,Z 131.937,A -85,B 0,C 180,E1 -21462.312,E2 -21462.312} C_VEL
LIN {X 0,Y 199.609,Z 131.926,A -85,B 0,C 180,E1 -21465.239,E2 -21465.239} C_VEL
LIN {X 0,Y 199.631,Z 131.925,A -85,B 0,C 180,E1 -21468.02,E2 -21468.02} C_VEL
LIN {X 0,Y 199.675,Z 131.925,A -85,B 0,C 180,E1 -21470.745,E2 -21470.745} C_VEL
LIN {X 0,Y 199.633,Z 131.926,A -85,B 0,C 180,E1 -21475.719,E2 -21475.719} C_VEL
LIN {X 0,Y 199.703,Z 131.921,A -85,B 0,C 180,E1 -21478.139,E2 -21478.139} C_VEL
LIN {X 0,Y 199.687,Z 131.919,A -85,B 0,C 180,E1 -21482.773,E2 -21482.773} C_VEL
LIN {X 0,Y 199.75,Z 131.911,A -85,B 0,C 180,E1 -21487.232,E2 -21487.232} C_VEL
LIN {X 0,Y 199.838,Z 131.904,A -85,B 0,C 180,E1 -21491.723,E2 -21491.723} C_VEL
LIN {X 0,Y 199.837,Z 131.897,A -85,B 0,C 180,E1 -21495.75,E2 -21495.75} C_VEL
LIN {X 0,Y 200.076,Z 131.875,A -85,B 0,C 180,E1 -21499.886,E2 -21499.886} C_VEL
LIN {X 0,Y 200.133,Z 131.863,A -85,B 0,C 180,E1 -21501.927,E2 -21501.927} C_VEL
LIN {X 0,Y 200.323,Z 131.842,A -85,B 0,C 180,E1 -21507.991,E2 -21507.991} C_VEL
LIN {X 0,Y 200.481,Z 131.825,A -85,B 0,C 180,E1 -21510.001,E2 -21510.001} C_VEL
LIN {X 0,Y 200.032,Z 131.865,A -85,B 0,C 180,E1 -21514.031,E2 -21514.031} C_VEL
LIN {X 0,Y 200.134,Z 131.871,A -85,B 0,C 180,E1 -21518.076,E2 -21518.076} C_VEL
LIN {X 0,Y 199.917,Z 131.886,A -85,B 0,C 180,E1 -21522.178,E2 -21522.178} C_VEL
LIN {X 0,Y 199.808,Z 131.907,A -85,B 0,C 180,E1 -21526.345,E2 -21526.345} C_VEL
LIN {X 0,Y 199.703,Z 131.921,A -85,B 0,C 180,E1 -21530.606,E2 -21530.606} C_VEL
LIN {X 0,Y 199.676,Z 131.925,A -85,B 0,C 180,E1 -21534.985,E2 -21534.985} C_VEL
LIN {X 0,Y 199.678,Z 131.929,A -85,B 0,C 180,E1 -21539.523,E2 -21539.523} C_VEL
LIN {X 0,Y 199.697,Z 132.079,A -85,B 0,C 180,E1 -21542.412,E2 -21542.412} C_VEL
LIN {X 0,Y 200.787,Z 134.963,A -85,B 0,C 180,E1 -21542.873,E2 -21542.873} C_VEL
LIN {X 0,Y 202.173,Z 137.195,A -85,B 0,C 180,E1 -21543.339,E2 -21543.339} C_VEL
LIN {X 0,Y 210.183,Z 151.653,A -85,B 0,C 180,E1 -21546,E2 -21546} C_VEL
LIN {X 0,Y 220.032,Z 170.506,A -85,B 0,C 180,E1 -21549.044,E2 -21549.044} C_VEL
LIN {X 0,Y 231.754,Z 194.232,A -85,B 0,C 180,E1 -21552.362,E2 -21552.362} C_VEL
LIN {X 0,Y 235.788,Z 202.754,A -85,B 0,C 180,E1 -21553.441,E2 -21553.441} C_VEL
LIN {X 0,Y 224.738,Z 311.935,A -85,B 0,C 180,E1 -21558.676,E2 -21558.676} C_VEL
LIN {X 0,Y 222.606,Z 330.495,A -85,B 0,C 180,E1 -21559.964,E2 -21559.964} C_VEL
LIN {X 0,Y 219.984,Z 348.698,A -85,B 0,C 180,E1 -21561.612,E2 -21561.612} C_VEL
LIN {X 0,Y 217.233,Z 365.499,A -85,B 0,C 180,E1 -21563.525,E2 -21563.525} C_VEL
LIN {X 0,Y 214.096,Z 381.976,A -85,B 0,C 180,E1 -21565.823,E2 -21565.823} C_VEL
LIN {X 0,Y 211.059,Z 397.011,A -85,B 0,C 180,E1 -21568.368,E2 -21568.368} C_VEL
LIN {X 0,Y 208.072,Z 411.338,A -85,B 0,C 180,E1 -21571.284,E2 -21571.284} C_VEL
LIN {X 0,Y 205.215,Z 425.154,A -85,B 0,C 180,E1 -21574.654,E2 -21574.654} C_VEL
LIN {X 0,Y 203.097,Z 435.414,A -85,B 0,C 180,E1 -21577.626,E2 -21577.626} C_VEL
LIN {X 0,Y 201.193,Z 445.799,A -85,B 0,C 180,E1 -21581.13,E2 -21581.13} C_VEL
LIN {X 0,Y 199.726,Z 454.83,A -85,B 0,C 180,E1 -21584.698,E2 -21584.698} C_VEL
LIN {X 0,Y 198.644,Z 463.418,A -85,B 0,C 180,E1 -21588.779,E2 -21588.779} C_VEL
LIN {X 0,Y 198.04,Z 470.701,A -85,B 0,C 180,E1 -21592.967,E2 -21592.967} C_VEL
LIN {X 0,Y 197.883,Z 476.374,A -85,B 0,C 180,E1 -21596.946,E2 -21596.946} C_VEL
LIN {X 0,Y 197.998,Z 481.022,A -85,B 0,C 180,E1 -21601.017,E2 -21601.017} C_VEL
LIN {X 0,Y 198.454,Z 483.844,A -85,B 0,C 180,E1 -21604.061,E2 -21604.061} C_VEL
LIN {X 0,Y 199.281,Z 486.686,A -85,B 0,C 180,E1 -21608.109,E2 -21608.109} C_VEL
LIN {X 0,Y 201.001,Z 488.688,A -85,B 0,C 180,E1 -21612.11,E2 -21612.11} C_VEL
LIN {X 0,Y 204.935,Z 490.076,A -85,B 0,C 180,E1 -21617.977,E2 -21617.977} C_VEL
LIN {X 0,Y 210.805,Z 489.618,A -85,B 0,C 180,E1 -21623.582,E2 -21623.582} C_VEL
LIN {X 0,Y 215.843,Z 488.309,A -85,B 0,C 180,E1 -21627.119,E2 -21627.119} C_VEL
LIN {X 0,Y 225.022,Z 484.994,A -85,B 0,C 180,E1 -21632.069,E2 -21632.069} C_VEL
LIN {X 0,Y 234.696,Z 480.678,A -85,B 0,C 180,E1 -21636.047,E2 -21636.047} C_VEL
LIN {X 0,Y 246.573,Z 474.607,A -85,B 0,C 180,E1 -21639.889,E2 -21639.889} C_VEL
LIN {X 0,Y 255.187,Z 469.802,A -85,B 0,C 180,E1 -21642.167,E2 -21642.167} C_VEL
LIN {X 0,Y 256.24,Z 469.32,A -85,B 0,C 180,E1 -21642.747,E2 -21642.747} C_VEL
LIN {X 0,Y 248.005,Z 475.339,A -85,B 0,C 180,E1 -21644.615,E2 -21644.615} C_VEL
LIN {X 0,Y 244.017,Z 478.103,A -85,B 0,C 180,E1 -21645.414,E2 -21645.414} C_VEL
LIN {X 0,Y 229.011,Z 486.953,A -85,B 0,C 180,E1 -21647.673,E2 -21647.673} C_VEL
LIN {X 0,Y 225.235,Z 489.181,A -85,B 0,C 180,E1 -21648.652,E2 -21648.652} C_VEL
LIN {X 0,Y 216.611,Z 494.599,A -85,B 0,C 180,E1 -21651.941,E2 -21651.941} C_VEL
LIN {X 0,Y 206.789,Z 500.841,A -85,B 0,C 180,E1 -21657.057,E2 -21657.057} C_VEL
LIN {X 0,Y 201.412,Z 504.183,A -85,B 0,C 180,E1 -21660.756,E2 -21660.756} C_VEL
LIN {X 0,Y 195.432,Z 507.91,A -85,B 0,C 180,E1 -21666.697,E2 -21666.697} C_VEL
LIN {X 0,Y 192.457,Z 509.769,A -85,B 0,C 180,E1 -21671.703,E2 -21671.703} C_VEL
LIN {X 0,Y 190.842,Z 510.402,A -85,B 0,C 180,E1 -21677.233,E2 -21677.233} C_VEL
LIN {X 0,Y 190.723,Z 509.989,A -85,B 0,C 180,E1 -21681.523,E2 -21681.523} C_VEL
LIN {X 0,Y 191.311,Z 508.556,A -85,B 0,C 180,E1 -21685.785,E2 -21685.785} C_VEL
LIN {X 0,Y 191.883,Z 506.048,A -85,B 0,C 180,E1 -21689.999,E2 -21689.999} C_VEL
LIN {X 0,Y 191.783,Z 502.067,A -85,B 0,C 180,E1 -21694.202,E2 -21694.202} C_VEL
LIN {X 0,Y 191.684,Z 498.12,A -85,B 0,C 180,E1 -21697.386,E2 -21697.386} C_VEL
LIN {X 0,Y 191.662,Z 491.515,A -85,B 0,C 180,E1 -21701.634,E2 -21701.634} C_VEL
LIN {X 0,Y 192.187,Z 484.44,A -85,B 0,C 180,E1 -21705.373,E2 -21705.373} C_VEL
LIN {X 0,Y 193.406,Z 474.585,A -85,B 0,C 180,E1 -21709.64,E2 -21709.64} C_VEL
LIN {X 0,Y 195.097,Z 464.236,A -85,B 0,C 180,E1 -21713.343,E2 -21713.343} C_VEL
LIN {X 0,Y 197.514,Z 452.117,A -85,B 0,C 180,E1 -21716.967,E2 -21716.967} C_VEL
LIN {X 0,Y 200.101,Z 439.875,A -85,B 0,C 180,E1 -21720.031,E2 -21720.031} C_VEL
LIN {X 0,Y 203.287,Z 425.729,A -85,B 0,C 180,E1 -21722.989,E2 -21722.989} C_VEL
LIN {X 0,Y 206.573,Z 410.406,A -85,B 0,C 180,E1 -21725.634,E2 -21725.634} C_VEL
LIN {X 0,Y 209.991,Z 393.902,A -85,B 0,C 180,E1 -21727.948,E2 -21727.948} C_VEL
LIN {X 0,Y 213.371,Z 375.796,A -85,B 0,C 180,E1 -21729.961,E2 -21729.961} C_VEL
LIN {X 0,Y 216.125,Z 359.236,A -85,B 0,C 180,E1 -21731.394,E2 -21731.394} C_VEL
LIN {X 0,Y 218.395,Z 341.332,A -85,B 0,C 180,E1 -21732.592,E2 -21732.592} C_VEL
LIN {X 0,Y 231.6,Z 218.74,A -85,B 0,C 180,E1 -21738.658,E2 -21738.658} C_VEL
LIN {X 0,Y 222.621,Z 197.142,A -85,B 0,C 180,E1 -21741.356,E2 -21741.356} C_VEL
LIN {X 0,Y 212.141,Z 173.29,A -85,B 0,C 180,E1 -21744.741,E2 -21744.741} C_VEL
LIN {X 0,Y 202.201,Z 152.198,A -85,B 0,C 180,E1 -21748.211,E2 -21748.211} C_VEL
LIN {X 0,Y 194.63,Z 137.228,A -85,B 0,C 180,E1 -21751.042,E2 -21751.042} C_VEL
LIN {X 0,Y 192.817,Z 133.653,A -85,B 0,C 180,E1 -21751.791,E2 -21751.791} C_VEL
LIN {X 0,Y 192.641,Z 132.807,A -85,B 0,C 180,E1 -21752.133,E2 -21752.133} C_VEL
LIN {X 0,Y 192.702,Z 132.796,A -85,B 0,C 180,E1 -21756.348,E2 -21756.348} C_VEL
LIN {X 0,Y 192.728,Z 132.793,A -85,B 0,C 180,E1 -21761.457,E2 -21761.457} C_VEL
LIN {X 0,Y 192.768,Z 132.785,A -85,B 0,C 180,E1 -21765.214,E2 -21765.214} C_VEL
LIN {X 0,Y 193.016,Z 132.75,A -85,B 0,C 180,E1 -21769.511,E2 -21769.511} C_VEL
LIN {X 0,Y 193.001,Z 132.747,A -85,B 0,C 180,E1 -21773.729,E2 -21773.729} C_VEL
LIN {X 0,Y 193.261,Z 132.724,A -85,B 0,C 180,E1 -21777.916,E2 -21777.916} C_VEL
LIN {X 0,Y 193.443,Z 132.7,A -85,B 0,C 180,E1 -21780,E2 -21780} C_VEL
LIN {X 0,Y 192.977,Z 132.758,A -85,B 0,C 180,E1 -21784.177,E2 -21784.177} C_VEL
LIN {X 0,Y 193.076,Z 132.746,A -85,B 0,C 180,E1 -21788.372,E2 -21788.372} C_VEL
LIN {X 0,Y 192.85,Z 132.771,A -85,B 0,C 180,E1 -21792.63,E2 -21792.63} C_VEL
LIN {X 0,Y 192.754,Z 132.782,A -85,B 0,C 180,E1 -21796.959,E2 -21796.959} C_VEL
LIN {X 0,Y 192.633,Z 132.802,A -85,B 0,C 180,E1 -21801.398,E2 -21801.398} C_VEL
LIN {X 0,Y 192.661,Z 132.789,A -85,B 0,C 180,E1 -21804.225,E2 -21804.225} C_VEL
LIN {X 0,Y 192.647,Z 132.8,A -85,B 0,C 180,E1 -21808.893,E2 -21808.893} C_VEL
LIN {X 0,Y 192.596,Z 132.805,A -85,B 0,C 180,E1 -21813.187,E2 -21813.187} C_VEL
LIN {X 0,Y 192.548,Z 132.805,A -85,B 0,C 180,E1 -21818.353,E2 -21818.353} C_VEL
LIN {X 0,Y 192.514,Z 132.816,A -85,B 0,C 180,E1 -21823.105,E2 -21823.105} C_VEL
LIN {X 0,Y 192.55,Z 132.804,A -85,B 0,C 180,E1 -21826.886,E2 -21826.886} C_VEL
LIN {X 0,Y 192.597,Z 132.803,A -85,B 0,C 180,E1 -21831.661,E2 -21831.661} C_VEL
LIN {X 0,Y 192.599,Z 132.807,A -85,B 0,C 180,E1 -21836.816,E2 -21836.816} C_VEL
LIN {X 0,Y 192.664,Z 132.788,A -85,B 0,C 180,E1 -21841.693,E2 -21841.693} C_VEL
LIN {X 0,Y 192.711,Z 132.792,A -85,B 0,C 180,E1 -21846.351,E2 -21846.351} C_VEL
LIN {X 0,Y 192.782,Z 132.782,A -85,B 0,C 180,E1 -21851.415,E2 -21851.415} C_VEL
LIN {X 0,Y 192.823,Z 132.777,A -85,B 0,C 180,E1 -21857.369,E2 -21857.369} C_VEL
LIN {X 0,Y 193.021,Z 132.753,A -85,B 0,C 180,E1 -21859.512,E2 -21859.512} C_VEL
LIN {X 0,Y 193.005,Z 132.756,A -85,B 0,C 180,E1 -21863.73,E2 -21863.73} C_VEL
LIN {X 0,Y 193.265,Z 132.721,A -85,B 0,C 180,E1 -21867.917,E2 -21867.917} C_VEL
LIN {X 0,Y 193.445,Z 132.701,A -85,B 0,C 180,E1 -21870.001,E2 -21870.001} C_VEL
LIN {X 0,Y 192.979,Z 132.743,A -85,B 0,C 180,E1 -21874.178,E2 -21874.178} C_VEL
LIN {X 0,Y 193.081,Z 132.748,A -85,B 0,C 180,E1 -21878.373,E2 -21878.373} C_VEL
LIN {X 0,Y 192.856,Z 132.767,A -85,B 0,C 180,E1 -21882.631,E2 -21882.631} C_VEL
LIN {X 0,Y 192.761,Z 132.783,A -85,B 0,C 180,E1 -21886.96,E2 -21886.96} C_VEL
LIN {X 0,Y 192.64,Z 132.801,A -85,B 0,C 180,E1 -21891.398,E2 -21891.398} C_VEL
LIN {X 0,Y 192.667,Z 132.793,A -85,B 0,C 180,E1 -21894.226,E2 -21894.226} C_VEL
LIN {X 0,Y 192.653,Z 132.8,A -85,B 0,C 180,E1 -21898.893,E2 -21898.893} C_VEL
LIN {X 0,Y 192.616,Z 132.803,A -85,B 0,C 180,E1 -21900.872,E2 -21900.872} C_VEL
LIN {X 0,Y 193.773,Z 135.865,A -85,B 0,C 180,E1 -21901.426,E2 -21901.426} C_VEL
LIN {X 0,Y 195.055,Z 137.9,A -85,B 0,C 180,E1 -21901.877,E2 -21901.877} C_VEL
LIN {X 0,Y 204.202,Z 154.269,A -85,B 0,C 180,E1 -21905.058,E2 -21905.058} C_VEL
LIN {X 0,Y 215.083,Z 175.299,A -85,B 0,C 180,E1 -21908.547,E2 -21908.547} C_VEL
LIN {X 0,Y 226.497,Z 198.712,A -85,B 0,C 180,E1 -21911.889,E2 -21911.889} C_VEL
LIN {X 0,Y 229.437,Z 205.008,A -85,B 0,C 180,E1 -21912.7,E2 -21912.7} C_VEL
LIN {X 0,Y 218.057,Z 312.699,A -85,B 0,C 180,E1 -21918.027,E2 -21918.027} C_VEL
LIN {X 0,Y 216.052,Z 329.913,A -85,B 0,C 180,E1 -21919.261,E2 -21919.261} C_VEL
LIN {X 0,Y 213.36,Z 348.288,A -85,B 0,C 180,E1 -21920.952,E2 -21920.952} C_VEL
LIN {X 0,Y 210.364,Z 366.049,A -85,B 0,C 180,E1 -21923.033,E2 -21923.033} C_VEL
LIN {X 0,Y 207.16,Z 382.338,A -85,B 0,C 180,E1 -21925.371,E2 -21925.371} C_VEL
LIN {X 0,Y 204.045,Z 397.53,A -85,B 0,C 180,E1 -21928.024,E2 -21928.024} C_VEL
LIN {X 0,Y 200.843,Z 412.464,A -85,B 0,C 180,E1 -21931.181,E2 -21931.181} C_VEL
LIN {X 0,Y 197.906,Z 426.536,A -85,B 0,C 180,E1 -21934.777,E2 -21934.777} C_VEL
LIN {X 0,Y 195.474,Z 438.326,A -85,B 0,C 180,E1 -21938.375,E2 -21938.375} C_VEL
LIN {X 0,Y 193.471,Z 449.729,A -85,B 0,C 180,E1 -21942.561,E2 -21942.561} C_VEL
LIN {X 0,Y 191.991,Z 459.253,A -85,B 0,C 180,E1 -21946.774,E2 -21946.774} C_VEL
LIN {X 0,Y 191.275,Z 466.277,A -85,B 0,C 180,E1 -21950.483,E2 -21950.483} C_VEL
LIN {X 0,Y 190.782,Z 473.138,A -85,B 0,C 180,E1 -21954.787,E2 -21954.787} C_VEL
LIN {X 0,Y 190.821,Z 478.464,A -85,B 0,C 180,E1 -21958.945,E2 -21958.945} C_VEL
LIN {X 0,Y 191.058,Z 481.835,A -85,B 0,C 180,E1 -21962.108,E2 -21962.108} C_VEL
LIN {X 0,Y 191.772,Z 485.402,A -85,B 0,C 180,E1 -21966.312,E2 -21966.312} C_VEL
LIN {X 0,Y 193.198,Z 488.26,A -85,B 0,C 180,E1 -21970.825,E2 -21970.825} C_VEL
LIN {X 0,Y 196.631,Z 490.446,A -85,B 0,C 180,E1 -21976.615,E2 -21976.615} C_VEL
LIN {X 0,Y 202.13,Z 490.988,A -85,B 0,C 180,E1 -21982.486,E2 -21982.486} C_VEL
LIN {X 0,Y 209.694,Z 489.796,A -85,B 0,C 180,E1 -21987.983,E2 -21987.983} C_VEL
LIN {X 0,Y 219.276,Z 486.947,A -85,B 0,C 180,E1 -21993.015,E2 -21993.015} C_VEL
LIN {X 0,Y 230.777,Z 482.469,A -85,B 0,C 180,E1 -21997.522,E2 -21997.522} C_VEL
LIN {X 0,Y 243.926,Z 476.432,A -85,B 0,C 180,E1 -22001.504,E2 -22001.504} C_VEL
LIN {X 0,Y 246.737,Z 475.022,A -85,B 0,C 180,E1 -22002.238,E2 -22002.238} C_VEL
LIN {X 0,Y 246.395,Z 475.396,A -85,B 0,C 180,E1 -22002.75,E2 -22002.75} C_VEL
LIN {X 0,Y 233.18,Z 484.09,A -85,B 0,C 180,E1 -22006.113,E2 -22006.113} C_VEL
LIN {X 0,Y 225.235,Z 489.181,A -85,B 0,C 180,E1 -22008.652,E2 -22008.652} C_VEL
LIN {X 0,Y 221.496,Z 491.357,A -85,B 0,C 180,E1 -22009.696,E2 -22009.696} C_VEL
LIN {X 0,Y 208.537,Z 497.309,A -85,B 0,C 180,E1 -22012.541,E2 -22012.541} C_VEL
LIN {X 0,Y 204.944,Z 498.962,A -85,B 0,C 180,E1 -22013.743,E2 -22013.743} C_VEL
LIN {X 0,Y 203.984,Z 499.441,A -85,B 0,C 180,E1 -22014.2,E2 -22014.2} C_VEL
LIN {X 0,Y 195.035,Z 504.336,A -85,B 0,C 180,E1 -22019.862,E2 -22019.862} C_VEL
LIN {X 0,Y 188.828,Z 507.573,A -85,B 0,C 180,E1 -22025.831,E2 -22025.831} C_VEL
LIN {X 0,Y 185.08,Z 509.299,A -85,B 0,C 180,E1 -22032.314,E2 -22032.314} C_VEL
LIN {X 0,Y 183.882,Z 509.517,A -85,B 0,C 180,E1 -22036.741,E2 -22036.741} C_VEL
LIN {X 0,Y 183.959,Z 508.225,A -85,B 0,C 180,E1 -22043.417,E2 -22043.417} C_VEL
LIN {X 0,Y 184.301,Z 507.28,A -85,B 0,C 180,E1 -22045.625,E2 -22045.625} C_VEL
LIN {X 0,Y 184.933,Z 504.575,A -85,B 0,C 180,E1 -22049.999,E2 -22049.999} C_VEL
LIN {X 0,Y 184.83,Z 501.555,A -85,B 0,C 180,E1 -22053.268,E2 -22053.268} C_VEL
LIN {X 0,Y 184.776,Z 497.739,A -85,B 0,C 180,E1 -22056.551,E2 -22056.551} C_VEL
LIN {X 0,Y 184.651,Z 491.24,A -85,B 0,C 180,E1 -22060.969,E2 -22060.969} C_VEL
LIN {X 0,Y 185.105,Z 484.265,A -85,B 0,C 180,E1 -22064.848,E2 -22064.848} C_VEL
LIN {X 0,Y 186.294,Z 474.211,A -85,B 0,C 180,E1 -22069.416,E2 -22069.416} C_VEL
LIN {X 0,Y 188.182,Z 462.747,A -85,B 0,C 180,E1 -22073.669,E2 -22073.669} C_VEL
LIN {X 0,Y 190.499,Z 451.401,A -85,B 0,C 180,E1 -22077.157,E2 -22077.157} C_VEL
LIN {X 0,Y 193.376,Z 438.106,A -85,B 0,C 180,E1 -22080.583,E2 -22080.583} C_VEL
LIN {X 0,Y 196.649,Z 423.783,A -85,B 0,C 180,E1 -22083.637,E2 -22083.637} C_VEL
LIN {X 0,Y 200.102,Z 407.903,A -85,B 0,C 180,E1 -22086.41,E2 -22086.41} C_VEL
LIN {X 0,Y 203.206,Z 393.234,A -85,B 0,C 180,E1 -22088.5,E2 -22088.5} C_VEL
LIN {X 0,Y 206.457,Z 376.317,A -85,B 0,C 180,E1 -22090.457,E2 -22090.457} C_VEL
LIN {X 0,Y 209.611,Z 357.91,A -85,B 0,C 180,E1 -22092.11,E2 -22092.11} C_VEL
LIN {X 0,Y 211.939,Z 339.827,A -85,B 0,C 180,E1 -22093.346,E2 -22093.346} C_VEL
LIN {X 0,Y 225.218,Z 220.593,A -85,B 0,C 180,E1 -22099.444,E2 -22099.444} C_VEL
LIN {X 0,Y 215.851,Z 197.945,A -85,B 0,C 180,E1 -22102.375,E2 -22102.375} C_VEL
LIN {X 0,Y 205.155,Z 173.673,A -85,B 0,C 180,E1 -22105.98,E2 -22105.98} C_VEL
LIN {X 0,Y 196.634,Z 155.565,A -85,B 0,C 180,E1 -22109.092,E2 -22109.092} C_VEL
LIN {X 0,Y 189.379,Z 141.085,A -85,B 0,C 180,E1 -22111.911,E2 -22111.911} C_VEL
LIN {X 0,Y 187.185,Z 137.34,A -85,B 0,C 180,E1 -22112.769,E2 -22112.769} C_VEL
LIN {X 0,Y 185.847,Z 134.932,A -85,B 0,C 180,E1 -22113.317,E2 -22113.317} C_VEL
LIN {X 0,Y 185.556,Z 133.689,A -85,B 0,C 180,E1 -22113.5,E2 -22113.5} C_VEL
LIN {X 0,Y 185.593,Z 133.685,A -85,B 0,C 180,E1 -22117.748,E2 -22117.748} C_VEL
LIN {X 0,Y 185.686,Z 133.664,A -85,B 0,C 180,E1 -22122.375,E2 -22122.375} C_VEL
LIN {X 0,Y 185.761,Z 133.65,A -85,B 0,C 180,E1 -22126.88,E2 -22126.88} C_VEL
LIN {X 0,Y 186.025,Z 133.627,A -85,B 0,C 180,E1 -22131.308,E2 -22131.308} C_VEL
LIN {X 0,Y 186.205,Z 133.602,A -85,B 0,C 180,E1 -22137.837,E2 -22137.837} C_VEL
LIN {X 0,Y 186.406,Z 133.577,A -85,B 0,C 180,E1 -22140,E2 -22140} C_VEL
LIN {X 0,Y 185.924,Z 133.637,A -85,B 0,C 180,E1 -22144.336,E2 -22144.336} C_VEL
LIN {X 0,Y 186.026,Z 133.625,A -85,B 0,C 180,E1 -22148.692,E2 -22148.692} C_VEL
LIN {X 0,Y 185.761,Z 133.656,A -85,B 0,C 180,E1 -22153.121,E2 -22153.121} C_VEL
LIN {X 0,Y 185.687,Z 133.661,A -85,B 0,C 180,E1 -22157.625,E2 -22157.625} C_VEL
LIN {X 0,Y 185.593,Z 133.676,A -85,B 0,C 180,E1 -22162.252,E2 -22162.252} C_VEL
LIN {X 0,Y 185.559,Z 133.683,A -85,B 0,C 180,E1 -22167.033,E2 -22167.033} C_VEL
LIN {X 0,Y 185.576,Z 133.677,A -85,B 0,C 180,E1 -22169.494,E2 -22169.494} C_VEL
LIN {X 0,Y 185.496,Z 133.691,A -85,B 0,C 180,E1 -22174.633,E2 -22174.633} C_VEL
LIN {X 0,Y 185.502,Z 133.684,A -85,B 0,C 180,E1 -22177.314,E2 -22177.314} C_VEL
LIN {X 0,Y 185.468,Z 133.691,A -85,B 0,C 180,E1 -22180.726,E2 -22180.726} C_VEL
LIN {X 0,Y 185.508,Z 133.68,A -85,B 0,C 180,E1 -22186.039,E2 -22186.039} C_VEL
LIN {X 0,Y 185.527,Z 133.686,A -85,B 0,C 180,E1 -22189.913,E2 -22189.913} C_VEL
LIN {X 0,Y 185.558,Z 133.677,A -85,B 0,C 180,E1 -22192.701,E2 -22192.701} C_VEL
LIN {X 0,Y 185.544,Z 133.684,A -85,B 0,C 180,E1 -22197.977,E2 -22197.977} C_VEL
LIN {X 0,Y 185.581,Z 133.673,A -85,B 0,C 180,E1 -22200.577,E2 -22200.577} C_VEL
LIN {X 0,Y 185.605,Z 133.677,A -85,B 0,C 180,E1 -22205.387,E2 -22205.387} C_VEL
LIN {X 0,Y 185.71,Z 133.664,A -85,B 0,C 180,E1 -22211.102,E2 -22211.102} C_VEL
LIN {X 0,Y 185.743,Z 133.659,A -85,B 0,C 180,E1 -22216.88,E2 -22216.88} C_VEL
LIN {X 0,Y 186.03,Z 133.618,A -85,B 0,C 180,E1 -22221.31,E2 -22221.31} C_VEL
LIN {X 0,Y 186.209,Z 133.599,A -85,B 0,C 180,E1 -22227.838,E2 -22227.838} C_VEL
LIN {X 0,Y 186.408,Z 133.578,A -85,B 0,C 180,E1 -22230.001,E2 -22230.001} C_VEL
LIN {X 0,Y 185.927,Z 133.621,A -85,B 0,C 180,E1 -22234.337,E2 -22234.337} C_VEL
LIN {X 0,Y 186.031,Z 133.626,A -85,B 0,C 180,E1 -22238.693,E2 -22238.693} C_VEL
LIN {X 0,Y 185.768,Z 133.653,A -85,B 0,C 180,E1 -22243.122,E2 -22243.122} C_VEL
LIN {X 0,Y 185.693,Z 133.658,A -85,B 0,C 180,E1 -22247.626,E2 -22247.626} C_VEL
LIN {X 0,Y 185.6,Z 133.673,A -85,B 0,C 180,E1 -22252.252,E2 -22252.252} C_VEL
LIN {X 0,Y 185.566,Z 133.678,A -85,B 0,C 180,E1 -22257.033,E2 -22257.033} C_VEL
LIN {X 0,Y 185.607,Z 133.881,A -85,B 0,C 180,E1 -22259.353,E2 -22259.353} C_VEL
LIN {X 0,Y 186.798,Z 136.88,A -85,B 0,C 180,E1 -22259.903,E2 -22259.903} C_VEL
LIN {X 0,Y 188.079,Z 138.853,A -85,B 0,C 180,E1 -22260.374,E2 -22260.374} C_VEL
LIN {X 0,Y 198.153,Z 156.82,A -85,B 0,C 180,E1 -22264.062,E2 -22264.062} C_VEL
LIN {X 0,Y 209.309,Z 178.515,A -85,B 0,C 180,E1 -22267.792,E2 -22267.792} C_VEL
LIN {X 0,Y 220.93,Z 202.486,A -85,B 0,C 180,E1 -22271.307,E2 -22271.307} C_VEL
LIN {X 0,Y 222.964,Z 206.904,A -85,B 0,C 180,E1 -22271.896,E2 -22271.896} C_VEL
LIN {X 0,Y 213.581,Z 292.581,A -85,B 0,C 180,E1 -22276.208,E2 -22276.208} C_VEL
LIN {X 0,Y 211.161,Z 316.368,A -85,B 0,C 180,E1 -22277.579,E2 -22277.579} C_VEL
LIN {X 0,Y 208.84,Z 334.507,A -85,B 0,C 180,E1 -22278.987,E2 -22278.987} C_VEL
LIN {X 0,Y 206.048,Z 351.909,A -85,B 0,C 180,E1 -22280.718,E2 -22280.718} C_VEL
LIN {X 0,Y 203.234,Z 367.809,A -85,B 0,C 180,E1 -22282.691,E2 -22282.691} C_VEL
LIN {X 0,Y 199.942,Z 384.178,A -85,B 0,C 180,E1 -22285.166,E2 -22285.166} C_VEL
LIN {X 0,Y 196.753,Z 399.126,A -85,B 0,C 180,E1 -22287.904,E2 -22287.904} C_VEL
LIN {X 0,Y 193.749,Z 412.981,A -85,B 0,C 180,E1 -22290.946,E2 -22290.946} C_VEL
LIN {X 0,Y 190.963,Z 426.011,A -85,B 0,C 180,E1 -22294.378,E2 -22294.378} C_VEL
LIN {X 0,Y 188.472,Z 437.906,A -85,B 0,C 180,E1 -22298.106,E2 -22298.106} C_VEL
LIN {X 0,Y 186.637,Z 448.118,A -85,B 0,C 180,E1 -22301.901,E2 -22301.901} C_VEL
LIN {X 0,Y 185.016,Z 457.981,A -85,B 0,C 180,E1 -22306.266,E2 -22306.266} C_VEL
LIN {X 0,Y 184.248,Z 465.354,A -85,B 0,C 180,E1 -22310.116,E2 -22310.116} C_VEL
LIN {X 0,Y 183.69,Z 472.907,A -85,B 0,C 180,E1 -22314.928,E2 -22314.928} C_VEL
LIN {X 0,Y 183.751,Z 478.013,A -85,B 0,C 180,E1 -22318.904,E2 -22318.904} C_VEL
LIN {X 0,Y 184.13,Z 482.61,A -85,B 0,C 180,E1 -22323.282,E2 -22323.282} C_VEL
LIN {X 0,Y 184.72,Z 485.399,A -85,B 0,C 180,E1 -22326.554,E2 -22326.554} C_VEL
LIN {X 0,Y 187.144,Z 489.386,A -85,B 0,C 180,E1 -22333.022,E2 -22333.022} C_VEL
LIN {X 0,Y 191.529,Z 491.489,A -85,B 0,C 180,E1 -22339.284,E2 -22339.284} C_VEL
LIN {X 0,Y 195.634,Z 491.894,A -85,B 0,C 180,E1 -22343.276,E2 -22343.276} C_VEL
LIN {X 0,Y 200.647,Z 491.614,A -85,B 0,C 180,E1 -22347.087,E2 -22347.087} C_VEL
LIN {X 0,Y 210.075,Z 489.749,A -85,B 0,C 180,E1 -22352.362,E2 -22352.362} C_VEL
LIN {X 0,Y 221.306,Z 486.343,A -85,B 0,C 180,E1 -22357.112,E2 -22357.112} C_VEL
LIN {X 0,Y 234.374,Z 481.385,A -85,B 0,C 180,E1 -22361.276,E2 -22361.276} C_VEL
LIN {X 0,Y 238.034,Z 479.856,A -85,B 0,C 180,E1 -22362.426,E2 -22362.426} C_VEL
LIN {X 0,Y 225.703,Z 487.16,A -85,B 0,C 180,E1 -22365.647,E2 -22365.647} C_VEL
LIN {X 0,Y 213.05,Z 494.334,A -85,B 0,C 180,E1 -22369.963,E2 -22369.963} C_VEL
LIN {X 0,Y 203.984,Z 499.441,A -85,B 0,C 180,E1 -22374.2,E2 -22374.2} C_VEL
LIN {X 0,Y 200.812,Z 500.943,A -85,B 0,C 180,E1 -22375.553,E2 -22375.553} C_VEL
LIN {X 0,Y 194.317,Z 503.128,A -85,B 0,C 180,E1 -22377.636,E2 -22377.636} C_VEL
LIN {X 0,Y 188.165,Z 504.878,A -85,B 0,C 180,E1 -22379.89,E2 -22379.89} C_VEL
LIN {X 0,Y 185.596,Z 505.712,A -85,B 0,C 180,E1 -22381.49,E2 -22381.49} C_VEL
LIN {X 0,Y 180.639,Z 507.785,A -85,B 0,C 180,E1 -22387.102,E2 -22387.102} C_VEL
LIN {X 0,Y 178.254,Z 508.515,A -85,B 0,C 180,E1 -22391.613,E2 -22391.613} C_VEL
LIN {X 0,Y 176.943,Z 508.476,A -85,B 0,C 180,E1 -22396.211,E2 -22396.211} C_VEL
LIN {X 0,Y 176.701,Z 507.66,A -85,B 0,C 180,E1 -22400.844,E2 -22400.844} C_VEL
LIN {X 0,Y 177.303,Z 505.937,A -85,B 0,C 180,E1 -22405.452,E2 -22405.452} C_VEL
LIN {X 0,Y 177.671,Z 504.64,A -85,B 0,C 180,E1 -22407.732,E2 -22407.732} C_VEL
LIN {X 0,Y 177.991,Z 503.013,A -85,B 0,C 180,E1 -22409.998,E2 -22409.998} C_VEL
LIN {X 0,Y 177.876,Z 498.627,A -85,B 0,C 180,E1 -22414.531,E2 -22414.531} C_VEL
LIN {X 0,Y 177.738,Z 494.47,A -85,B 0,C 180,E1 -22417.827,E2 -22417.827} C_VEL
LIN {X 0,Y 177.819,Z 487.12,A -85,B 0,C 180,E1 -22422.553,E2 -22422.553} C_VEL
LIN {X 0,Y 178.615,Z 478.257,A -85,B 0,C 180,E1 -22427.162,E2 -22427.162} C_VEL
LIN {X 0,Y 179.901,Z 468.831,A -85,B 0,C 180,E1 -22431.182,E2 -22431.182} C_VEL
LIN {X 0,Y 181.959,Z 457.758,A -85,B 0,C 180,E1 -22435.14,E2 -22435.14} C_VEL
LIN {X 0,Y 184.756,Z 444.892,A -85,B 0,C 180,E1 -22438.967,E2 -22438.967} C_VEL
LIN {X 0,Y 187.71,Z 431.605,A -85,B 0,C 180,E1 -22442.242,E2 -22442.242} C_VEL
LIN {X 0,Y 190.917,Z 417.578,A -85,B 0,C 180,E1 -22445.111,E2 -22445.111} C_VEL
LIN {X 0,Y 194.668,Z 401.109,A -85,B 0,C 180,E1 -22447.859,E2 -22447.859} C_VEL
LIN {X 0,Y 198.157,Z 383.911,A -85,B 0,C 180,E1 -22450.168,E2 -22450.168} C_VEL
LIN {X 0,Y 201.454,Z 366.359,A -85,B 0,C 180,E1 -22452.017,E2 -22452.017} C_VEL
LIN {X 0,Y 204.29,Z 348.29,A -85,B 0,C 180,E1 -22453.473,E2 -22453.473} C_VEL
LIN {X 0,Y 207.132,Z 322.635,A -85,B 0,C 180,E1 -22455.012,E2 -22455.012} C_VEL
LIN {X 0,Y 218.752,Z 222.279,A -85,B 0,C 180,E1 -22460.266,E2 -22460.266} C_VEL
LIN {X 0,Y 210.125,Z 201.27,A -85,B 0,C 180,E1 -22463.079,E2 -22463.079} C_VEL
LIN {X 0,Y 199.672,Z 177.313,A -85,B 0,C 180,E1 -22466.744,E2 -22466.744} C_VEL
LIN {X 0,Y 191.494,Z 159.775,A -85,B 0,C 180,E1 -22469.845,E2 -22469.845} C_VEL
LIN {X 0,Y 184.563,Z 145.705,A -85,B 0,C 180,E1 -22472.657,E2 -22472.657} C_VEL
LIN {X 0,Y 180.005,Z 138.077,A -85,B 0,C 180,E1 -22474.489,E2 -22474.489} C_VEL
LIN {X 0,Y 178.763,Z 135.629,A -85,B 0,C 180,E1 -22475.047,E2 -22475.047} C_VEL
LIN {X 0,Y 178.552,Z 134.563,A -85,B 0,C 180,E1 -22475.219,E2 -22475.219} C_VEL
LIN {X 0,Y 178.646,Z 134.546,A -85,B 0,C 180,E1 -22481.656,E2 -22481.656} C_VEL
LIN {X 0,Y 178.684,Z 134.535,A -85,B 0,C 180,E1 -22486.35,E2 -22486.35} C_VEL
LIN {X 0,Y 178.974,Z 134.505,A -85,B 0,C 180,E1 -22490.963,E2 -22490.963} C_VEL
LIN {X 0,Y 179.151,Z 134.479,A -85,B 0,C 180,E1 -22497.752,E2 -22497.752} C_VEL
LIN {X 0,Y 179.369,Z 134.454,A -85,B 0,C 180,E1 -22500,E2 -22500} C_VEL
LIN {X 0,Y 178.873,Z 134.515,A -85,B 0,C 180,E1 -22504.507,E2 -22504.507} C_VEL
LIN {X 0,Y 178.975,Z 134.504,A -85,B 0,C 180,E1 -22509.037,E2 -22509.037} C_VEL
LIN {X 0,Y 178.684,Z 134.541,A -85,B 0,C 180,E1 -22513.65,E2 -22513.65} C_VEL
LIN {X 0,Y 178.646,Z 134.539,A -85,B 0,C 180,E1 -22518.344,E2 -22518.344} C_VEL
LIN {X 0,Y 178.508,Z 134.555,A -85,B 0,C 180,E1 -22523.186,E2 -22523.186} C_VEL
LIN {X 0,Y 178.484,Z 134.563,A -85,B 0,C 180,E1 -22528.198,E2 -22528.198} C_VEL
LIN {X 0,Y 178.476,Z 134.557,A -85,B 0,C 180,E1 -22530.791,E2 -22530.791} C_VEL
LIN {X 0,Y 178.482,Z 134.564,A -85,B 0,C 180,E1 -22534.221,E2 -22534.221} C_VEL
LIN {X 0,Y 178.392,Z 134.567,A -85,B 0,C 180,E1 -22539.075,E2 -22539.075} C_VEL
LIN {X 0,Y 178.406,Z 134.573,A -85,B 0,C 180,E1 -22542.043,E2 -22542.043} C_VEL
LIN {X 0,Y 178.424,Z 134.564,A -85,B 0,C 180,E1 -22545.154,E2 -22545.154} C_VEL
LIN {X 0,Y 178.439,Z 134.565,A -85,B 0,C 180,E1 -22548.446,E2 -22548.446} C_VEL
LIN {X 0,Y 178.485,Z 134.561,A -85,B 0,C 180,E1 -22551.954,E2 -22551.954} C_VEL
LIN {X 0,Y 178.49,Z 134.562,A -85,B 0,C 180,E1 -22556.549,E2 -22556.549} C_VEL
LIN {X 0,Y 178.522,Z 134.557,A -85,B 0,C 180,E1 -22560.008,E2 -22560.008} C_VEL
LIN {X 0,Y 178.534,Z 134.559,A -85,B 0,C 180,E1 -22564.877,E2 -22564.877} C_VEL
LIN {X 0,Y 178.654,Z 134.543,A -85,B 0,C 180,E1 -22570.757,E2 -22570.757} C_VEL
LIN {X 0,Y 178.667,Z 134.536,A -85,B 0,C 180,E1 -22576.35,E2 -22576.35} C_VEL
LIN {X 0,Y 178.978,Z 134.496,A -85,B 0,C 180,E1 -22580.965,E2 -22580.965} C_VEL
LIN {X 0,Y 179.155,Z 134.477,A -85,B 0,C 180,E1 -22587.753,E2 -22587.753} C_VEL
LIN {X 0,Y 179.371,Z 134.454,A -85,B 0,C 180,E1 -22590.001,E2 -22590.001} C_VEL
LIN {X 0,Y 178.875,Z 134.499,A -85,B 0,C 180,E1 -22594.508,E2 -22594.508} C_VEL
LIN {X 0,Y 178.981,Z 134.504,A -85,B 0,C 180,E1 -22599.038,E2 -22599.038} C_VEL
LIN {X 0,Y 178.69,Z 134.537,A -85,B 0,C 180,E1 -22603.651,E2 -22603.651} C_VEL
LIN {X 0,Y 178.653,Z 134.533,A -85,B 0,C 180,E1 -22608.345,E2 -22608.345} C_VEL
LIN {X 0,Y 178.514,Z 134.552,A -85,B 0,C 180,E1 -22613.186,E2 -22613.186} C_VEL
LIN {X 0,Y 178.57,Z 134.548,A -85,B 0,C 180,E1 -22617.626,E2 -22617.626} C_VEL
LIN {X 0,Y 179.681,Z 137.521,A -85,B 0,C 180,E1 -22618.207,E2 -22618.207} C_VEL
LIN {X 0,Y 180.926,Z 139.431,A -85,B 0,C 180,E1 -22618.699,E2 -22618.699} C_VEL
LIN {X 0,Y 189.648,Z 155.008,A -85,B 0,C 180,E1 -22622.125,E2 -22622.125} C_VEL
LIN {X 0,Y 197.469,Z 169.713,A -85,B 0,C 180,E1 -22624.946,E2 -22624.946} C_VEL
LIN {X 0,Y 208.483,Z 191.743,A -85,B 0,C 180,E1 -22628.603,E2 -22628.603} C_VEL
LIN {X 0,Y 216.567,Z 208.901,A -85,B 0,C 180,E1 -22631.084,E2 -22631.084} C_VEL
LIN {X 0,Y 207.282,Z 291.119,A -85,B 0,C 180,E1 -22635.36,E2 -22635.36} C_VEL
LIN {X 0,Y 204.574,Z 316.421,A -85,B 0,C 180,E1 -22636.853,E2 -22636.853} C_VEL
LIN {X 0,Y 202.152,Z 334.81,A -85,B 0,C 180,E1 -22638.325,E2 -22638.325} C_VEL
LIN {X 0,Y 199.116,Z 353.229,A -85,B 0,C 180,E1 -22640.227,E2 -22640.227} C_VEL
LIN {X 0,Y 195.999,Z 370.212,A -85,B 0,C 180,E1 -22642.441,E2 -22642.441} C_VEL
LIN {X 0,Y 192.403,Z 387.33,A -85,B 0,C 180,E1 -22645.198,E2 -22645.198} C_VEL
LIN {X 0,Y 188.936,Z 403.047,A -85,B 0,C 180,E1 -22648.303,E2 -22648.303} C_VEL
LIN {X 0,Y 185.657,Z 417.486,A -85,B 0,C 180,E1 -22651.759,E2 -22651.759} C_VEL
LIN {X 0,Y 183.263,Z 429.012,A -85,B 0,C 180,E1 -22655.049,E2 -22655.049} C_VEL
LIN {X 0,Y 180.95,Z 440.152,A -85,B 0,C 180,E1 -22658.776,E2 -22658.776} C_VEL
LIN {X 0,Y 179.079,Z 450.482,A -85,B 0,C 180,E1 -22662.882,E2 -22662.882} C_VEL
LIN {X 0,Y 177.631,Z 460.023,A -85,B 0,C 180,E1 -22667.431,E2 -22667.431} C_VEL
LIN {X 0,Y 176.912,Z 468.023,A -85,B 0,C 180,E1 -22672.007,E2 -22672.007} C_VEL
LIN {X 0,Y 176.626,Z 474.655,A -85,B 0,C 180,E1 -22676.578,E2 -22676.578} C_VEL
LIN {X 0,Y 176.779,Z 480.007,A -85,B 0,C 180,E1 -22681.139,E2 -22681.139} C_VEL
LIN {X 0,Y 177.281,Z 483.345,A -85,B 0,C 180,E1 -22684.547,E2 -22684.547} C_VEL
LIN {X 0,Y 178.922,Z 488.11,A -85,B 0,C 180,E1 -22690.883,E2 -22690.883} C_VEL
LIN {X 0,Y 181.552,Z 490.609,A -85,B 0,C 180,E1 -22695.722,E2 -22695.722} C_VEL
LIN {X 0,Y 184.847,Z 492.089,A -85,B 0,C 180,E1 -22700.01,E2 -22700.01} C_VEL
LIN {X 0,Y 191.666,Z 492.859,A -85,B 0,C 180,E1 -22706.104,E2 -22706.104} C_VEL
LIN {X 0,Y 197.488,Z 492.464,A -85,B 0,C 180,E1 -22709.882,E2 -22709.882} C_VEL
LIN {X 0,Y 207.924,Z 490.557,A -85,B 0,C 180,E1 -22715.072,E2 -22715.072} C_VEL
LIN {X 0,Y 220.302,Z 487.127,A -85,B 0,C 180,E1 -22719.645,E2 -22719.645} C_VEL
LIN {X 0,Y 224.766,Z 485.641,A -85,B 0,C 180,E1 -22721.043,E2 -22721.043} C_VEL
LIN {X 0,Y 228.335,Z 484.515,A -85,B 0,C 180,E1 -22722.377,E2 -22722.377} C_VEL
LIN {X 0,Y 214.166,Z 491.895,A -85,B 0,C 180,E1 -22726.437,E2 -22726.437} C_VEL
LIN {X 0,Y 205.679,Z 496.145,A -85,B 0,C 180,E1 -22729.515,E2 -22729.515} C_VEL
LIN {X 0,Y 194.969,Z 501.401,A -85,B 0,C 180,E1 -22734.776,E2 -22734.776} C_VEL
LIN {X 0,Y 188.499,Z 504.407,A -85,B 0,C 180,E1 -22739.04,E2 -22739.04} C_VEL
LIN {X 0,Y 185.596,Z 505.712,A -85,B 0,C 180,E1 -22741.49,E2 -22741.49} C_VEL
LIN {X 0,Y 183.21,Z 506.487,A -85,B 0,C 180,E1 -22743.153,E2 -22743.153} C_VEL
LIN {X 0,Y 178.006,Z 507.28,A -85,B 0,C 180,E1 -22745.816,E2 -22745.816} C_VEL
LIN {X 0,Y 174.048,Z 507.519,A -85,B 0,C 180,E1 -22748.051,E2 -22748.051} C_VEL
LIN {X 0,Y 171.996,Z 507.594,A -85,B 0,C 180,E1 -22749.884,E2 -22749.884} C_VEL
LIN {X 0,Y 171.602,Z 507.609,A -85,B 0,C 180,E1 -22750.527,E2 -22750.527} C_VEL
LIN {X 0,Y 170.025,Z 507.431,A -85,B 0,C 180,E1 -22755.639,E2 -22755.639} C_VEL
LIN {X 0,Y 169.714,Z 506.404,A -85,B 0,C 180,E1 -22760.464,E2 -22760.464} C_VEL
LIN {X 0,Y 170.334,Z 504.462,A -85,B 0,C 180,E1 -22765.265,E2 -22765.265} C_VEL
LIN {X 0,Y 170.755,Z 503.107,A -85,B 0,C 180,E1 -22767.64,E2 -22767.64} C_VEL
LIN {X 0,Y 171.06,Z 501.426,A -85,B 0,C 180,E1 -22769.998,E2 -22769.998} C_VEL
LIN {X 0,Y 170.952,Z 496.74,A -85,B 0,C 180,E1 -22774.715,E2 -22774.715} C_VEL
LIN {X 0,Y 170.714,Z 491.4,A -85,B 0,C 180,E1 -22778.874,E2 -22778.874} C_VEL
LIN {X 0,Y 171.022,Z 483.702,A -85,B 0,C 180,E1 -22783.666,E2 -22783.666} C_VEL
LIN {X 0,Y 171.836,Z 475.484,A -85,B 0,C 180,E1 -22787.862,E2 -22787.862} C_VEL
LIN {X 0,Y 173.25,Z 465.746,A -85,B 0,C 180,E1 -22792.037,E2 -22792.037} C_VEL
LIN {X 0,Y 175.478,Z 454.316,A -85,B 0,C 180,E1 -22796.138,E2 -22796.138} C_VEL
LIN {X 0,Y 178.254,Z 441.881,A -85,B 0,C 180,E1 -22799.844,E2 -22799.844} C_VEL
LIN {X 0,Y 181.674,Z 427.162,A -85,B 0,C 180,E1 -22803.451,E2 -22803.451} C_VEL
LIN {X 0,Y 185.097,Z 412.54,A -85,B 0,C 180,E1 -22806.387,E2 -22806.387} C_VEL
LIN {X 0,Y 188.668,Z 396.75,A -85,B 0,C 180,E1 -22808.979,E2 -22808.979} C_VEL
LIN {X 0,Y 192.124,Z 380.077,A -85,B 0,C 180,E1 -22811.18,E2 -22811.18} C_VEL
LIN {X 0,Y 195.499,Z 361.706,A -85,B 0,C 180,E1 -22813.079,E2 -22813.079} C_VEL
LIN {X 0,Y 198.16,Z 344.152,A -85,B 0,C 180,E1 -22814.462,E2 -22814.462} C_VEL
LIN {X 0,Y 211.213,Z 234.036,A -85,B 0,C 180,E1 -22820.583,E2 -22820.583} C_VEL
LIN {X 0,Y 212.337,Z 224.011,A -85,B 0,C 180,E1 -22821.11,E2 -22821.11} C_VEL
LIN {X 0,Y 203.073,Z 201.408,A -85,B 0,C 180,E1 -22824.267,E2 -22824.267} C_VEL
LIN {X 0,Y 193.711,Z 179.962,A -85,B 0,C 180,E1 -22827.702,E2 -22827.702} C_VEL
LIN {X 0,Y 186.328,Z 163.848,A -85,B 0,C 180,E1 -22830.637,E2 -22830.637} C_VEL
LIN {X 0,Y 179.572,Z 150.055,A -85,B 0,C 180,E1 -22833.477,E2 -22833.477} C_VEL
LIN {X 0,Y 175.002,Z 142.4,A -85,B 0,C 180,E1 -22835.395,E2 -22835.395} C_VEL
LIN {X 0,Y 173.298,Z 139.372,A -85,B 0,C 180,E1 -22836.155,E2 -22836.155} C_VEL
LIN {X 0,Y 171.808,Z 136.917,A -85,B 0,C 180,E1 -22836.814,E2 -22836.814} C_VEL
LIN {X 0,Y 171.453,Z 135.444,A -85,B 0,C 180,E1 -22837.082,E2 -22837.082} C_VEL
LIN {X 0,Y 171.575,Z 135.428,A -85,B 0,C 180,E1 -22840.872,E2 -22840.872} C_VEL
LIN {X 0,Y 171.606,Z 135.419,A -85,B 0,C 180,E1 -22845.776,E2 -22845.776} C_VEL
LIN {X 0,Y 171.906,Z 135.385,A -85,B 0,C 180,E1 -22850.588,E2 -22850.588} C_VEL
LIN {X 0,Y 171.821,Z 135.377,A -85,B 0,C 180,E1 -22855.308,E2 -22855.308} C_VEL
LIN {X 0,Y 172.331,Z 135.33,A -85,B 0,C 180,E1 -22860,E2 -22860} C_VEL
LIN {X 0,Y 171.823,Z 135.393,A -85,B 0,C 180,E1 -22864.693,E2 -22864.693} C_VEL
LIN {X 0,Y 171.907,Z 135.384,A -85,B 0,C 180,E1 -22869.412,E2 -22869.412} C_VEL
LIN {X 0,Y 171.606,Z 135.421,A -85,B 0,C 180,E1 -22874.225,E2 -22874.225} C_VEL
LIN {X 0,Y 171.541,Z 135.429,A -85,B 0,C 180,E1 -22879.563,E2 -22879.563} C_VEL
LIN {X 0,Y 171.466,Z 135.435,A -85,B 0,C 180,E1 -22885.617,E2 -22885.617} C_VEL
LIN {X 0,Y 171.439,Z 135.434,A -85,B 0,C 180,E1 -22890.588,E2 -22890.588} C_VEL
LIN {X 0,Y 171.389,Z 135.45,A -85,B 0,C 180,E1 -22895.036,E2 -22895.036} C_VEL
LIN {X 0,Y 171.354,Z 135.442,A -85,B 0,C 180,E1 -22898.809,E2 -22898.809} C_VEL
LIN {X 0,Y 171.341,Z 135.452,A -85,B 0,C 180,E1 -22904.211,E2 -22904.211} C_VEL
LIN {X 0,Y 171.373,Z 135.449,A -85,B 0,C 180,E1 -22908.995,E2 -22908.995} C_VEL
LIN {X 0,Y 171.433,Z 135.44,A -85,B 0,C 180,E1 -22912.055,E2 -22912.055} C_VEL
LIN {X 0,Y 171.418,Z 135.444,A -85,B 0,C 180,E1 -22917.794,E2 -22917.794} C_VEL
LIN {X 0,Y 171.448,Z 135.433,A -85,B 0,C 180,E1 -22920.536,E2 -22920.536} C_VEL
LIN {X 0,Y 171.465,Z 135.439,A -85,B 0,C 180,E1 -22925.805,E2 -22925.805} C_VEL
LIN {X 0,Y 171.61,Z 135.421,A -85,B 0,C 180,E1 -22930.877,E2 -22930.877} C_VEL
LIN {X 0,Y 171.585,Z 135.415,A -85,B 0,C 180,E1 -22935.775,E2 -22935.775} C_VEL
LIN {X 0,Y 171.905,Z 135.378,A -85,B 0,C 180,E1 -22940.59,E2 -22940.59} C_VEL
LIN {X 0,Y 171.826,Z 135.393,A -85,B 0,C 180,E1 -22945.309,E2 -22945.309} C_VEL
LIN {X 0,Y 172.334,Z 135.33,A -85,B 0,C 180,E1 -22950.002,E2 -22950.002} C_VEL
LIN {X 0,Y 171.825,Z 135.378,A -85,B 0,C 180,E1 -22954.694,E2 -22954.694} C_VEL
LIN {X 0,Y 171.913,Z 135.382,A -85,B 0,C 180,E1 -22959.413,E2 -22959.413} C_VEL
LIN {X 0,Y 171.613,Z 135.423,A -85,B 0,C 180,E1 -22964.226,E2 -22964.226} C_VEL
LIN {X 0,Y 171.547,Z 135.424,A -85,B 0,C 180,E1 -22969.563,E2 -22969.563} C_VEL
LIN {X 0,Y 171.488,Z 135.545,A -85,B 0,C 180,E1 -22975.829,E2 -22975.829} C_VEL
LIN {X 0,Y 172.556,Z 138.405,A -85,B 0,C 180,E1 -22976.412,E2 -22976.412} C_VEL
LIN {X 0,Y 174.031,Z 140.48,A -85,B 0,C 180,E1 -22977.023,E2 -22977.023} C_VEL
LIN {X 0,Y 184.059,Z 158.283,A -85,B 0,C 180,E1 -22981.159,E2 -22981.159} C_VEL
LIN {X 0,Y 192.443,Z 174.302,A -85,B 0,C 180,E1 -22984.319,E2 -22984.319} C_VEL
LIN {X 0,Y 202.908,Z 195.404,A -85,B 0,C 180,E1 -22987.919,E2 -22987.919} C_VEL
LIN {X 0,Y 210.171,Z 210.895,A -85,B 0,C 180,E1 -22990.237,E2 -22990.237} C_VEL
LIN {X 0,Y 198.158,Z 314.949,A -85,B 0,C 180,E1 -22995.979,E2 -22995.979} C_VEL
LIN {X 0,Y 195.69,Z 333.672,A -85,B 0,C 180,E1 -22997.497,E2 -22997.497} C_VEL
LIN {X 0,Y 192.772,Z 351.089,A -85,B 0,C 180,E1 -22999.303,E2 -22999.303} C_VEL
LIN {X 0,Y 189.867,Z 366.877,A -85,B 0,C 180,E1 -23001.344,E2 -23001.344} C_VEL
LIN {X 0,Y 186.432,Z 383.161,A -85,B 0,C 180,E1 -23003.912,E2 -23003.912} C_VEL
LIN {X 0,Y 183.065,Z 398.314,A -85,B 0,C 180,E1 -23006.834,E2 -23006.834} C_VEL
LIN {X 0,Y 179.582,Z 413.536,A -85,B 0,C 180,E1 -23010.391,E2 -23010.391} C_VEL
LIN {X 0,Y 176.733,Z 426.528,A -85,B 0,C 180,E1 -23014.06,E2 -23014.06} C_VEL
LIN {X 0,Y 174.108,Z 438.766,A -85,B 0,C 180,E1 -23018.192,E2 -23018.192} C_VEL
LIN {X 0,Y 172.259,Z 448.715,A -85,B 0,C 180,E1 -23022.182,E2 -23022.182} C_VEL
LIN {X 0,Y 170.66,Z 458.649,A -85,B 0,C 180,E1 -23026.909,E2 -23026.909} C_VEL
LIN {X 0,Y 170.047,Z 465.029,A -85,B 0,C 180,E1 -23030.484,E2 -23030.484} C_VEL
LIN {X 0,Y 169.553,Z 472.239,A -85,B 0,C 180,E1 -23035.244,E2 -23035.244} C_VEL
LIN {X 0,Y 169.614,Z 476.808,A -85,B 0,C 180,E1 -23038.813,E2 -23038.813} C_VEL
LIN {X 0,Y 170.011,Z 481.915,A -85,B 0,C 180,E1 -23043.555,E2 -23043.555} C_VEL
LIN {X 0,Y 171.212,Z 486.815,A -85,B 0,C 180,E1 -23049.45,E2 -23049.45} C_VEL
LIN {X 0,Y 174.714,Z 490.913,A -85,B 0,C 180,E1 -23056.354,E2 -23056.354} C_VEL
LIN {X 0,Y 180.371,Z 493.205,A -85,B 0,C 180,E1 -23062.932,E2 -23062.932} C_VEL
LIN {X 0,Y 188.275,Z 493.842,A -85,B 0,C 180,E1 -23069.03,E2 -23069.03} C_VEL
LIN {X 0,Y 198.52,Z 492.887,A -85,B 0,C 180,E1 -23074.501,E2 -23074.501} C_VEL
LIN {X 0,Y 210.629,Z 490.468,A -85,B 0,C 180,E1 -23079.343,E2 -23079.343} C_VEL
LIN {X 0,Y 215.146,Z 489.279,A -85,B 0,C 180,E1 -23080.792,E2 -23080.792} C_VEL
LIN {X 0,Y 218.675,Z 488.515,A -85,B 0,C 180,E1 -23082.335,E2 -23082.335} C_VEL
LIN {X 0,Y 204.59,Z 494.909,A -85,B 0,C 180,E1 -23086.603,E2 -23086.603} C_VEL
LIN {X 0,Y 196.369,Z 498.525,A -85,B 0,C 180,E1 -23089.891,E2 -23089.891} C_VEL
LIN {X 0,Y 185.915,Z 502.864,A -85,B 0,C 180,E1 -23095.455,E2 -23095.455} C_VEL
LIN {X 0,Y 178.893,Z 505.533,A -85,B 0,C 180,E1 -23100.777,E2 -23100.777} C_VEL
LIN {X 0,Y 174.032,Z 507.096,A -85,B 0,C 180,E1 -23106.18,E2 -23106.18} C_VEL
LIN {X 0,Y 171.602,Z 507.609,A -85,B 0,C 180,E1 -23110.527,E2 -23110.527} C_VEL
LIN {X 0,Y 170.161,Z 507.57,A -85,B 0,C 180,E1 -23112.447,E2 -23112.447} C_VEL
LIN {X 0,Y 166.522,Z 506.818,A -85,B 0,C 180,E1 -23115.576,E2 -23115.576} C_VEL
LIN {X 0,Y 163.866,Z 505.854,A -85,B 0,C 180,E1 -23118.158,E2 -23118.158} C_VEL
LIN {X 0,Y 162.852,Z 505.003,A -85,B 0,C 180,E1 -23120.187,E2 -23120.187} C_VEL
LIN {X 0,Y 162.814,Z 504.732,A -85,B 0,C 180,E1 -23120.877,E2 -23120.877} C_VEL
LIN {X 0,Y 163.372,Z 502.96,A -85,B 0,C 180,E1 -23125.063,E2 -23125.063} C_VEL
LIN {X 0,Y 163.833,Z 501.472,A -85,B 0,C 180,E1 -23127.54,E2 -23127.54} C_VEL
LIN {X 0,Y 164.167,Z 499.667,A -85,B 0,C 180,E1 -23129.998,E2 -23129.998} C_VEL
LIN {X 0,Y 164.063,Z 496.141,A -85,B 0,C 180,E1 -23133.682,E2 -23133.682} C_VEL
LIN {X 0,Y 163.861,Z 491.711,A -85,B 0,C 180,E1 -23137.391,E2 -23137.391} C_VEL
LIN {X 0,Y 163.91,Z 484.329,A -85,B 0,C 180,E1 -23142.378,E2 -23142.378} C_VEL
LIN {X 0,Y 164.578,Z 476.457,A -85,B 0,C 180,E1 -23146.751,E2 -23146.751} C_VEL
LIN {X 0,Y 165.906,Z 466.723,A -85,B 0,C 180,E1 -23151.26,E2 -23151.26} C_VEL
LIN {X 0,Y 167.907,Z 455.95,A -85,B 0,C 180,E1 -23155.404,E2 -23155.404} C_VEL
LIN {X 0,Y 170.355,Z 444.86,A -85,B 0,C 180,E1 -23158.994,E2 -23158.994} C_VEL
LIN {X 0,Y 173.614,Z 430.858,A -85,B 0,C 180,E1 -23162.779,E2 -23162.779} C_VEL
LIN {X 0,Y 176.941,Z 417.036,A -85,B 0,C 180,E1 -23165.862,E2 -23165.862} C_VEL
LIN {X 0,Y 180.418,Z 402.391,A -85,B 0,C 180,E1 -23168.553,E2 -23168.553} C_VEL
LIN {X 0,Y 183.831,Z 386.803,A -85,B 0,C 180,E1 -23170.895,E2 -23170.895} C_VEL
LIN {X 0,Y 187.396,Z 369.069,A -85,B 0,C 180,E1 -23173.005,E2 -23173.005} C_VEL
LIN {X 0,Y 190.552,Z 350.857,A -85,B 0,C 180,E1 -23174.672,E2 -23174.672} C_VEL
LIN {X 0,Y 193.123,Z 330.971,A -85,B 0,C 180,E1 -23176.041,E2 -23176.041} C_VEL
LIN {X 0,Y 205.967,Z 225.736,A -85,B 0,C 180,E1 -23181.986,E2 -23181.986} C_VEL
LIN {X 0,Y 195.21,Z 199.582,A -85,B 0,C 180,E1 -23185.828,E2 -23185.828} C_VEL
LIN {X 0,Y 185.805,Z 178.056,A -85,B 0,C 180,E1 -23189.503,E2 -23189.503} C_VEL
LIN {X 0,Y 177.457,Z 160.117,A -85,B 0,C 180,E1 -23193.066,E2 -23193.066} C_VEL
LIN {X 0,Y 173.186,Z 151.918,A -85,B 0,C 180,E1 -23194.941,E2 -23194.941} C_VEL
LIN {X 0,Y 168.043,Z 143.352,A -85,B 0,C 180,E1 -23197.233,E2 -23197.233} C_VEL
LIN {X 0,Y 166.312,Z 140.327,A -85,B 0,C 180,E1 -23198.055,E2 -23198.055} C_VEL
LIN {X 0,Y 164.729,Z 137.63,A -85,B 0,C 180,E1 -23198.82,E2 -23198.82} C_VEL
LIN {X 0,Y 164.441,Z 136.314,A -85,B 0,C 180,E1 -23199.109,E2 -23199.109} C_VEL
LIN {X 0,Y 164.501,Z 136.302,A -85,B 0,C 180,E1 -23202.599,E2 -23202.599} C_VEL
LIN {X 0,Y 164.776,Z 136.261,A -85,B 0,C 180,E1 -23208.802,E2 -23208.802} C_VEL
LIN {X 0,Y 164.858,Z 136.26,A -85,B 0,C 180,E1 -23212.652,E2 -23212.652} C_VEL
LIN {X 0,Y 165.294,Z 136.207,A -85,B 0,C 180,E1 -23220,E2 -23220} C_VEL
LIN {X 0,Y 164.837,Z 136.26,A -85,B 0,C 180,E1 -23227.115,E2 -23227.115} C_VEL
LIN {X 0,Y 164.776,Z 136.266,A -85,B 0,C 180,E1 -23231.198,E2 -23231.198} C_VEL
LIN {X 0,Y 164.502,Z 136.299,A -85,B 0,C 180,E1 -23237.401,E2 -23237.401} C_VEL
LIN {X 0,Y 164.47,Z 136.31,A -85,B 0,C 180,E1 -23239.99,E2 -23239.99} C_VEL
LIN {X 0,Y 164.39,Z 136.318,A -85,B 0,C 180,E1 -23246.135,E2 -23246.135} C_VEL
LIN {X 0,Y 164.372,Z 136.312,A -85,B 0,C 180,E1 -23251.229,E2 -23251.229} C_VEL
LIN {X 0,Y 164.291,Z 136.328,A -85,B 0,C 180,E1 -23256.791,E2 -23256.791} C_VEL
LIN {X 0,Y 164.289,Z 136.326,A -85,B 0,C 180,E1 -23259.917,E2 -23259.917} C_VEL
LIN {X 0,Y 164.276,Z 136.333,A -85,B 0,C 180,E1 -23263.343,E2 -23263.343} C_VEL
LIN {X 0,Y 164.319,Z 136.318,A -85,B 0,C 180,E1 -23266.82,E2 -23266.82} C_VEL
LIN {X 0,Y 164.34,Z 136.326,A -85,B 0,C 180,E1 -23270.333,E2 -23270.333} C_VEL
LIN {X 0,Y 164.343,Z 136.314,A -85,B 0,C 180,E1 -23274.343,E2 -23274.343} C_VEL
LIN {X 0,Y 164.39,Z 136.318,A -85,B 0,C 180,E1 -23279.136,E2 -23279.136} C_VEL
LIN {X 0,Y 164.417,Z 136.318,A -85,B 0,C 180,E1 -23284.696,E2 -23284.696} C_VEL
LIN {X 0,Y 164.52,Z 136.298,A -85,B 0,C 180,E1 -23290.019,E2 -23290.019} C_VEL
LIN {X 0,Y 164.534,Z 136.293,A -85,B 0,C 180,E1 -23295.152,E2 -23295.152} C_VEL
LIN {X 0,Y 164.835,Z 136.261,A -85,B 0,C 180,E1 -23300.182,E2 -23300.182} C_VEL
LIN {X 0,Y 164.862,Z 136.259,A -85,B 0,C 180,E1 -23302.654,E2 -23302.654} C_VEL
LIN {X 0,Y 165.052,Z 136.233,A -85,B 0,C 180,E1 -23307.561,E2 -23307.561} C_VEL
LIN {X 0,Y 165.297,Z 136.207,A -85,B 0,C 180,E1 -23310.002,E2 -23310.002} C_VEL
LIN {X 0,Y 164.864,Z 136.263,A -85,B 0,C 180,E1 -23317.349,E2 -23317.349} C_VEL
